LIN {X 0,Y 599.988,Z 849.399,A -85,B 0,C 180,E1 26596.435,E2 26596.435} C_VEL
LIN {X 0,Y 597.537,Z 878.172,A -85,B 0,C 180,E1 26595.722,E2 26595.722} C_VEL
LIN {X 0,Y 595.265,Z 899.969,A -85,B 0,C 180,E1 26595.037,E2 26595.037} C_VEL
LIN {X 0,Y 592.79,Z 920.942,A -85,B 0,C 180,E1 26594.253,E2 26594.253} C_VEL
LIN {X 0,Y 590.222,Z 940.863,A -85,B 0,C 180,E1 26593.384,E2 26593.384} C_VEL
LIN {X 0,Y 587.234,Z 961.854,A -85,B 0,C 180,E1 26592.336,E2 26592.336} C_VEL
LIN {X 0,Y 583.301,Z 987.615,A -85,B 0,C 180,E1 26590.839,E2 26590.839} C_VEL
LIN {X 0,Y 579.885,Z 1008.289,A -85,B 0,C 180,E1 26589.448,E2 26589.448} C_VEL
LIN {X 0,Y 576.852,Z 1026.156,A -85,B 0,C 180,E1 26588.099,E2 26588.099} C_VEL
LIN {X 0,Y 574.033,Z 1042.219,A -85,B 0,C 180,E1 26586.749,E2 26586.749} C_VEL
LIN {X 0,Y 571.11,Z 1058.494,A -85,B 0,C 180,E1 26585.23,E2 26585.23} C_VEL
LIN {X 0,Y 568.193,Z 1074.819,A -85,B 0,C 180,E1 26583.542,E2 26583.542} C_VEL
LIN {X 0,Y 564.878,Z 1093.745,A -85,B 0,C 180,E1 26581.358,E2 26581.358} C_VEL
LIN {X 0,Y 561.877,Z 1111.065,A -85,B 0,C 180,E1 26579.065,E2 26579.065} C_VEL
LIN {X 0,Y 559.756,Z 1124.375,A -85,B 0,C 180,E1 26577.096,E2 26577.096} C_VEL
LIN {X 0,Y 557.748,Z 1137.63,A -85,B 0,C 180,E1 26574.915,E2 26574.915} C_VEL
LIN {X 0,Y 555.8,Z 1152.163,A -85,B 0,C 180,E1 26572.196,E2 26572.196} C_VEL
LIN {X 0,Y 554.441,Z 1163.606,A -85,B 0,C 180,E1 26569.708,E2 26569.708} C_VEL
LIN {X 0,Y 553.521,Z 1172.704,A -85,B 0,C 180,E1 26567.449,E2 26567.449} C_VEL
LIN {X 0,Y 552.864,Z 1180.922,A -85,B 0,C 180,E1 26565.095,E2 26565.095} C_VEL
LIN {X 0,Y 552.339,Z 1189.025,A -85,B 0,C 180,E1 26562.334,E2 26562.334} C_VEL
LIN {X 0,Y 552.078,Z 1195.294,A -85,B 0,C 180,E1 26559.591,E2 26559.591} C_VEL
LIN {X 0,Y 551.97,Z 1199.532,A -85,B 0,C 180,E1 26557.18,E2 26557.18} C_VEL
LIN {X 0,Y 551.918,Z 1202.669,A -85,B 0,C 180,E1 26554.676,E2 26554.676} C_VEL
LIN {X 0,Y 551.91,Z 1204.6,A -85,B 0,C 180,E1 26551.869,E2 26551.869} C_VEL
LIN {X 0,Y 551.895,Z 1204.872,A -85,B 0,C 180,E1 26549.377,E2 26549.377} C_VEL
LIN {X 0,Y 551.916,Z 1203.978,A -85,B 0,C 180,E1 26546.988,E2 26546.988} C_VEL
LIN {X 0,Y 551.93,Z 1201.872,A -85,B 0,C 180,E1 26544.595,E2 26544.595} C_VEL
LIN {X 0,Y 552,Z 1198.251,A -85,B 0,C 180,E1 26541.983,E2 26541.983} C_VEL
LIN {X 0,Y 552.17,Z 1192.609,A -85,B 0,C 180,E1 26539.145,E2 26539.145} C_VEL
LIN {X 0,Y 552.519,Z 1186.072,A -85,B 0,C 180,E1 26536.607,E2 26536.607} C_VEL
LIN {X 0,Y 552.999,Z 1178.8,A -85,B 0,C 180,E1 26534.264,E2 26534.264} C_VEL
LIN {X 0,Y 553.836,Z 1169.631,A -85,B 0,C 180,E1 26531.739,E2 26531.739} C_VEL
LIN {X 0,Y 555.152,Z 1157.326,A -85,B 0,C 180,E1 26528.887,E2 26528.887} C_VEL
LIN {X 0,Y 556.58,Z 1145.997,A -85,B 0,C 180,E1 26526.609,E2 26526.609} C_VEL
LIN {X 0,Y 558.321,Z 1133.823,A -85,B 0,C 180,E1 26524.432,E2 26524.432} C_VEL
LIN {X 0,Y 560.9,Z 1117.228,A -85,B 0,C 180,E1 26521.811,E2 26521.811} C_VEL
LIN {X 0,Y 563.604,Z 1100.917,A -85,B 0,C 180,E1 26519.567,E2 26519.567} C_VEL
LIN {X 0,Y 566.273,Z 1085.443,A -85,B 0,C 180,E1 26517.656,E2 26517.656} C_VEL
LIN {X 0,Y 569.654,Z 1066.711,A -85,B 0,C 180,E1 26515.586,E2 26515.586} C_VEL
LIN {X 0,Y 573.385,Z 1045.863,A -85,B 0,C 180,E1 26513.576,E2 26513.576} C_VEL
LIN {X 0,Y 576.391,Z 1028.822,A -85,B 0,C 180,E1 26512.115,E2 26512.115} C_VEL
LIN {X 0,Y 579.366,Z 1011.299,A -85,B 0,C 180,E1 26510.77,E2 26510.77} C_VEL
LIN {X 0,Y 582.452,Z 992.608,A -85,B 0,C 180,E1 26509.484,E2 26509.484} C_VEL
LIN {X 0,Y 585.633,Z 972.478,A -85,B 0,C 180,E1 26508.253,E2 26508.253} C_VEL
LIN {X 0,Y 589.484,Z 946.5,A -85,B 0,C 180,E1 26506.878,E2 26506.878} C_VEL
LIN {X 0,Y 592.403,Z 924.112,A -85,B 0,C 180,E1 26505.876,E2 26505.876} C_VEL
LIN {X 0,Y 594.962,Z 902.704,A -85,B 0,C 180,E1 26505.059,E2 26505.059} C_VEL
LIN {X 0,Y 597.166,Z 881.774,A -85,B 0,C 180,E1 26504.383,E2 26504.383} C_VEL
LIN {X 0,Y 599.156,Z 859.782,A -85,B 0,C 180,E1 26503.799,E2 26503.799} C_VEL
LIN {X 0,Y 601.177,Z 832.126,A -85,B 0,C 180,E1 26503.233,E2 26503.233} C_VEL
LIN {X 0,Y 602.837,Z 786.304,A -85,B 0,C 180,E1 26502.56,E2 26502.56} C_VEL
LIN {X 0,Y 609.733,Z 564.773,A -85,B 0,C 180,E1 26499.403,E2 26499.403} C_VEL
LIN {X 0,Y 614.382,Z 422.014,A -85,B 0,C 180,E1 26497.318,E2 26497.318} C_VEL
LIN {X 0,Y 602.713,Z 404.172,A -85,B 0,C 180,E1 26495.496,E2 26495.496} C_VEL
LIN {X 0,Y 590.418,Z 386.403,A -85,B 0,C 180,E1 26493.424,E2 26493.424} C_VEL
LIN {X 0,Y 579.878,Z 372.071,A -85,B 0,C 180,E1 26491.498,E2 26491.498} C_VEL
LIN {X 0,Y 572.08,Z 361.83,A -85,B 0,C 180,E1 26489.963,E2 26489.963} C_VEL
LIN {X 0,Y 567.6,Z 356.163,A -85,B 0,C 180,E1 26489.034,E2 26489.034} C_VEL
LIN {X 0,Y 563.365,Z 350.725,A -85,B 0,C 180,E1 26488.114,E2 26488.114} C_VEL
LIN {X 0,Y 559.96,Z 346.445,A -85,B 0,C 180,E1 26487.346,E2 26487.346} C_VEL
LIN {X 0,Y 557.435,Z 343.483,A -85,B 0,C 180,E1 26486.716,E2 26486.716} C_VEL
LIN {X 0,Y 555.888,Z 340.01,A -85,B 0,C 180,E1 26485.919,E2 26485.919} C_VEL
LIN {X 0,Y 553.761,Z 336.637,A -85,B 0,C 180,E1 26484.988,E2 26484.988} C_VEL
LIN {X 0,Y 553.461,Z 335.24,A -85,B 0,C 180,E1 26484.666,E2 26484.666} C_VEL
LIN {X 0,Y 553.477,Z 335.245,A -85,B 0,C 180,E1 26481.292,E2 26481.292} C_VEL
LIN {X 0,Y 553.497,Z 335.282,A -85,B 0,C 180,E1 26477.994,E2 26477.994} C_VEL
LIN {X 0,Y 553.448,Z 335.235,A -85,B 0,C 180,E1 26474.758,E2 26474.758} C_VEL
LIN {X 0,Y 553.503,Z 335.278,A -85,B 0,C 180,E1 26471.462,E2 26471.462} C_VEL
LIN {X 0,Y 553.449,Z 335.241,A -85,B 0,C 180,E1 26468.206,E2 26468.206} C_VEL
LIN {X 0,Y 553.46,Z 335.263,A -85,B 0,C 180,E1 26464.871,E2 26464.871} C_VEL
LIN {X 0,Y 553.478,Z 335.25,A -85,B 0,C 180,E1 26461.656,E2 26461.656} C_VEL
LIN {X 0,Y 553.437,Z 335.255,A -85,B 0,C 180,E1 26458.447,E2 26458.447} C_VEL
LIN {X 0,Y 553.498,Z 335.258,A -85,B 0,C 180,E1 26455.233,E2 26455.233} C_VEL
LIN {X 0,Y 553.429,Z 335.249,A -85,B 0,C 180,E1 26452.108,E2 26452.108} C_VEL
LIN {X 0,Y 553.481,Z 335.272,A -85,B 0,C 180,E1 26448.854,E2 26448.854} C_VEL
LIN {X 0,Y 553.424,Z 335.242,A -85,B 0,C 180,E1 26445.776,E2 26445.776} C_VEL
LIN {X 0,Y 553.45,Z 335.293,A -85,B 0,C 180,E1 26442.44,E2 26442.44} C_VEL
LIN {X 0,Y 553.434,Z 335.237,A -85,B 0,C 180,E1 26439.364,E2 26439.364} C_VEL
LIN {X 0,Y 553.421,Z 335.272,A -85,B 0,C 180,E1 26436.014,E2 26436.014} C_VEL
LIN {X 0,Y 553.44,Z 335.455,A -85,B 0,C 180,E1 26433.785,E2 26433.785} C_VEL
LIN {X 0,Y 554.447,Z 338.299,A -85,B 0,C 180,E1 26433.491,E2 26433.491} C_VEL
LIN {X 0,Y 556.848,Z 340.849,A -85,B 0,C 180,E1 26432.923,E2 26432.923} C_VEL
LIN {X 0,Y 558.75,Z 342.157,A -85,B 0,C 180,E1 26432.503,E2 26432.503} C_VEL
LIN {X 0,Y 560.898,Z 345.768,A -85,B 0,C 180,E1 26431.983,E2 26431.983} C_VEL
LIN {X 0,Y 564.13,Z 348.556,A -85,B 0,C 180,E1 26431.293,E2 26431.293} C_VEL
LIN {X 0,Y 566.949,Z 352.543,A -85,B 0,C 180,E1 26430.669,E2 26430.669} C_VEL
LIN {X 0,Y 569.277,Z 354.812,A -85,B 0,C 180,E1 26430.194,E2 26430.194} C_VEL
LIN {X 0,Y 572.686,Z 359.091,A -85,B 0,C 180,E1 26429.493,E2 26429.493} C_VEL
LIN {X 0,Y 574.265,Z 360.906,A -85,B 0,C 180,E1 26429.18,E2 26429.18} C_VEL
LIN {X 0,Y 578.146,Z 365.563,A -85,B 0,C 180,E1 26428.426,E2 26428.426} C_VEL
LIN {X 0,Y 584.331,Z 373.412,A -85,B 0,C 180,E1 26427.266,E2 26427.266} C_VEL
LIN {X 0,Y 591.597,Z 382.48,A -85,B 0,C 180,E1 26425.983,E2 26425.983} C_VEL
LIN {X 0,Y 603.802,Z 398.638,A -85,B 0,C 180,E1 26423.964,E2 26423.964} C_VEL
LIN {X 0,Y 614.272,Z 413.349,A -85,B 0,C 180,E1 26422.352,E2 26422.352} C_VEL
LIN {X 0,Y 607.005,Z 631.906,A -85,B 0,C 180,E1 26419.19,E2 26419.19} C_VEL
LIN {X 0,Y 603.673,Z 738.694,A -85,B 0,C 180,E1 26417.669,E2 26417.669} C_VEL
LIN {X 0,Y 602.74,Z 746.4,A -85,B 0,C 180,E1 26417.633,E2 26417.633} C_VEL
LIN {X 0,Y 597.897,Z 767.028,A -85,B 0,C 180,E1 26417.785,E2 26417.785} C_VEL
LIN {X 0,Y 597.208,Z 773.633,A -85,B 0,C 180,E1 26417.742,E2 26417.742} C_VEL
LIN {X 0,Y 595.598,Z 809.869,A -85,B 0,C 180,E1 26417.181,E2 26417.181} C_VEL
LIN {X 0,Y 593.757,Z 833.921,A -85,B 0,C 180,E1 26416.665,E2 26416.665} C_VEL
LIN {X 0,Y 591.733,Z 855.327,A -85,B 0,C 180,E1 26416.083,E2 26416.083} C_VEL
LIN {X 0,Y 589.538,Z 875.33,A -85,B 0,C 180,E1 26415.424,E2 26415.424} C_VEL
LIN {X 0,Y 586.99,Z 895.612,A -85,B 0,C 180,E1 26414.639,E2 26414.639} C_VEL
LIN {X 0,Y 583.725,Z 919.209,A -85,B 0,C 180,E1 26413.566,E2 26413.566} C_VEL
LIN {X 0,Y 579.717,Z 944.344,A -85,B 0,C 180,E1 26412.205,E2 26412.205} C_VEL
LIN {X 0,Y 576.363,Z 963.977,A -85,B 0,C 180,E1 26410.976,E2 26410.976} C_VEL
LIN {X 0,Y 573.108,Z 982.083,A -85,B 0,C 180,E1 26409.699,E2 26409.699} C_VEL
LIN {X 0,Y 569.76,Z 1000.085,A -85,B 0,C 180,E1 26408.277,E2 26408.277} C_VEL
LIN {X 0,Y 565.664,Z 1021.503,A -85,B 0,C 180,E1 26406.372,E2 26406.372} C_VEL
LIN {X 0,Y 561.8,Z 1041.554,A -85,B 0,C 180,E1 26404.327,E2 26404.327} C_VEL
LIN {X 0,Y 558.837,Z 1057.414,A -85,B 0,C 180,E1 26402.523,E2 26402.523} C_VEL
LIN {X 0,Y 555.913,Z 1073.578,A -85,B 0,C 180,E1 26400.478,E2 26400.478} C_VEL
LIN {X 0,Y 552.664,Z 1092.003,A -85,B 0,C 180,E1 26397.824,E2 26397.824} C_VEL
LIN {X 0,Y 550.501,Z 1105.479,A -85,B 0,C 180,E1 26395.612,E2 26395.612} C_VEL
LIN {X 0,Y 548.641,Z 1118.062,A -85,B 0,C 180,E1 26393.295,E2 26393.295} C_VEL
LIN {X 0,Y 546.895,Z 1131.586,A -85,B 0,C 180,E1 26390.438,E2 26390.438} C_VEL
LIN {X 0,Y 545.756,Z 1141.728,A -85,B 0,C 180,E1 26387.926,E2 26387.926} C_VEL
LIN {X 0,Y 545.016,Z 1149.714,A -85,B 0,C 180,E1 26385.645,E2 26385.645} C_VEL
LIN {X 0,Y 544.517,Z 1156.853,A -85,B 0,C 180,E1 26383.269,E2 26383.269} C_VEL
LIN {X 0,Y 544.153,Z 1163.946,A -85,B 0,C 180,E1 26380.374,E2 26380.374} C_VEL
LIN {X 0,Y 543.987,Z 1168.822,A -85,B 0,C 180,E1 26377.711,E2 26377.711} C_VEL
LIN {X 0,Y 543.928,Z 1172.048,A -85,B 0,C 180,E1 26375.274,E2 26375.274} C_VEL
LIN {X 0,Y 543.911,Z 1174.082,A -85,B 0,C 180,E1 26372.845,E2 26372.845} C_VEL
LIN {X 0,Y 543.907,Z 1174.974,A -85,B 0,C 180,E1 26370.105,E2 26370.105} C_VEL
LIN {X 0,Y 543.908,Z 1174.209,A -85,B 0,C 180,E1 26367.26,E2 26367.26} C_VEL
LIN {X 0,Y 543.924,Z 1172.26,A -85,B 0,C 180,E1 26364.832,E2 26364.832} C_VEL
LIN {X 0,Y 543.974,Z 1169.277,A -85,B 0,C 180,E1 26362.501,E2 26362.501} C_VEL
LIN {X 0,Y 544.103,Z 1164.965,A -85,B 0,C 180,E1 26360.053,E2 26360.053} C_VEL
LIN {X 0,Y 544.431,Z 1158.303,A -85,B 0,C 180,E1 26357.161,E2 26357.161} C_VEL
LIN {X 0,Y 544.968,Z 1150.36,A -85,B 0,C 180,E1 26354.463,E2 26354.463} C_VEL
LIN {X 0,Y 545.681,Z 1142.463,A -85,B 0,C 180,E1 26352.182,E2 26352.182} C_VEL
LIN {X 0,Y 546.677,Z 1133.331,A -85,B 0,C 180,E1 26349.889,E2 26349.889} C_VEL
LIN {X 0,Y 548.28,Z 1120.798,A -85,B 0,C 180,E1 26347.143,E2 26347.143} C_VEL
LIN {X 0,Y 550.321,Z 1106.606,A -85,B 0,C 180,E1 26344.495,E2 26344.495} C_VEL
LIN {X 0,Y 552.349,Z 1093.942,A -85,B 0,C 180,E1 26342.393,E2 26342.393} C_VEL
LIN {X 0,Y 554.911,Z 1079.043,A -85,B 0,C 180,E1 26340.178,E2 26340.178} C_VEL
LIN {X 0,Y 558.47,Z 1059.488,A -85,B 0,C 180,E1 26337.635,E2 26337.635} C_VEL
LIN {X 0,Y 561.504,Z 1043.16,A -85,B 0,C 180,E1 26335.758,E2 26335.758} C_VEL
LIN {X 0,Y 564.674,Z 1026.355,A -85,B 0,C 180,E1 26334.021,E2 26334.021} C_VEL
LIN {X 0,Y 568.677,Z 1005.892,A -85,B 0,C 180,E1 26332.114,E2 26332.114} C_VEL
LIN {X 0,Y 572.798,Z 983.808,A -85,B 0,C 180,E1 26330.338,E2 26330.338} C_VEL
LIN {X 0,Y 576.126,Z 965.309,A -85,B 0,C 180,E1 26329.022,E2 26329.022} C_VEL
LIN {X 0,Y 579.352,Z 946.439,A -85,B 0,C 180,E1 26327.829,E2 26327.829} C_VEL
LIN {X 0,Y 582.723,Z 925.413,A -85,B 0,C 180,E1 26326.66,E2 26326.66} C_VEL
LIN {X 0,Y 586.616,Z 898.562,A -85,B 0,C 180,E1 26325.394,E2 26325.394} C_VEL
LIN {X 0,Y 589.41,Z 876.434,A -85,B 0,C 180,E1 26324.525,E2 26324.525} C_VEL
LIN {X 0,Y 591.727,Z 855.412,A -85,B 0,C 180,E1 26323.83,E2 26323.83} C_VEL
LIN {X 0,Y 593.743,Z 834.118,A -85,B 0,C 180,E1 26323.251,E2 26323.251} C_VEL
LIN {X 0,Y 595.557,Z 810.404,A -85,B 0,C 180,E1 26322.74,E2 26322.74} C_VEL
LIN {X 0,Y 597.184,Z 774.353,A -85,B 0,C 180,E1 26322.178,E2 26322.178} C_VEL
LIN {X 0,Y 604.577,Z 550.918,A -85,B 0,C 180,E1 26318.968,E2 26318.968} C_VEL
LIN {X 0,Y 609.231,Z 417.375,A -85,B 0,C 180,E1 26317.008,E2 26317.008} C_VEL
LIN {X 0,Y 597.885,Z 401.698,A -85,B 0,C 180,E1 26315.209,E2 26315.209} C_VEL
LIN {X 0,Y 587.512,Z 387.83,A -85,B 0,C 180,E1 26313.435,E2 26313.435} C_VEL
LIN {X 0,Y 578.153,Z 376.088,A -85,B 0,C 180,E1 26311.719,E2 26311.719} C_VEL
LIN {X 0,Y 574.829,Z 371.978,A -85,B 0,C 180,E1 26311.077,E2 26311.077} C_VEL
LIN {X 0,Y 570.013,Z 366.1,A -85,B 0,C 180,E1 26310.112,E2 26310.112} C_VEL
LIN {X 0,Y 565.664,Z 360.778,A -85,B 0,C 180,E1 26309.201,E2 26309.201} C_VEL
LIN {X 0,Y 562.258,Z 356.818,A -85,B 0,C 180,E1 26308.464,E2 26308.464} C_VEL
LIN {X 0,Y 561.023,Z 355.163,A -85,B 0,C 180,E1 26308.184,E2 26308.184} C_VEL
LIN {X 0,Y 557.676,Z 351.854,A -85,B 0,C 180,E1 26307.438,E2 26307.438} C_VEL
LIN {X 0,Y 555.938,Z 349.05,A -85,B 0,C 180,E1 26307.01,E2 26307.01} C_VEL
LIN {X 0,Y 552.681,Z 346.292,A -85,B 0,C 180,E1 26306.253,E2 26306.253} C_VEL
LIN {X 0,Y 550.679,Z 342.754,A -85,B 0,C 180,E1 26305.719,E2 26305.719} C_VEL
LIN {X 0,Y 547.427,Z 340.512,A -85,B 0,C 180,E1 26304.928,E2 26304.928} C_VEL
LIN {X 0,Y 545.843,Z 337.847,A -85,B 0,C 180,E1 26304.481,E2 26304.481} C_VEL
LIN {X 0,Y 545.469,Z 336.245,A -85,B 0,C 180,E1 26304.33,E2 26304.33} C_VEL
LIN {X 0,Y 545.544,Z 336.224,A -85,B 0,C 180,E1 26301.166,E2 26301.166} C_VEL
LIN {X 0,Y 545.481,Z 336.282,A -85,B 0,C 180,E1 26297.936,E2 26297.936} C_VEL
LIN {X 0,Y 545.505,Z 336.221,A -85,B 0,C 180,E1 26294.586,E2 26294.586} C_VEL
LIN {X 0,Y 545.5,Z 336.281,A -85,B 0,C 180,E1 26291.525,E2 26291.525} C_VEL
LIN {X 0,Y 545.489,Z 336.226,A -85,B 0,C 180,E1 26288.114,E2 26288.114} C_VEL
LIN {X 0,Y 545.536,Z 336.265,A -85,B 0,C 180,E1 26285.047,E2 26285.047} C_VEL
LIN {X 0,Y 545.491,Z 336.229,A -85,B 0,C 180,E1 26281.786,E2 26281.786} C_VEL
LIN {X 0,Y 545.563,Z 336.252,A -85,B 0,C 180,E1 26278.635,E2 26278.635} C_VEL
LIN {X 0,Y 545.5,Z 336.235,A -85,B 0,C 180,E1 26275.374,E2 26275.374} C_VEL
LIN {X 0,Y 545.534,Z 336.236,A -85,B 0,C 180,E1 26272.099,E2 26272.099} C_VEL
LIN {X 0,Y 545.528,Z 336.251,A -85,B 0,C 180,E1 26268.904,E2 26268.904} C_VEL
LIN {X 0,Y 545.511,Z 336.224,A -85,B 0,C 180,E1 26265.565,E2 26265.565} C_VEL
LIN {X 0,Y 545.568,Z 336.274,A -85,B 0,C 180,E1 26262.288,E2 26262.288} C_VEL
LIN {X 0,Y 545.519,Z 336.229,A -85,B 0,C 180,E1 26258.946,E2 26258.946} C_VEL
LIN {X 0,Y 545.535,Z 336.344,A -85,B 0,C 180,E1 26256.906,E2 26256.906} C_VEL
LIN {X 0,Y 546.888,Z 339.751,A -85,B 0,C 180,E1 26256.053,E2 26256.053} C_VEL
LIN {X 0,Y 548.427,Z 341.539,A -85,B 0,C 180,E1 26255.437,E2 26255.437} C_VEL
LIN {X 0,Y 549.416,Z 343.962,A -85,B 0,C 180,E1 26254.939,E2 26254.939} C_VEL
LIN {X 0,Y 553.071,Z 348.19,A -85,B 0,C 180,E1 26254.026,E2 26254.026} C_VEL
LIN {X 0,Y 557.925,Z 354.223,A -85,B 0,C 180,E1 26252.864,E2 26252.864} C_VEL
LIN {X 0,Y 562.346,Z 359.743,A -85,B 0,C 180,E1 26251.859,E2 26251.859} C_VEL
LIN {X 0,Y 567.765,Z 366.71,A -85,B 0,C 180,E1 26250.686,E2 26250.686} C_VEL
LIN {X 0,Y 574.835,Z 376.016,A -85,B 0,C 180,E1 26249.243,E2 26249.243} C_VEL
LIN {X 0,Y 584.56,Z 389.121,A -85,B 0,C 180,E1 26247.397,E2 26247.397} C_VEL
LIN {X 0,Y 597.209,Z 407.344,A -85,B 0,C 180,E1 26245.185,E2 26245.185} C_VEL
LIN {X 0,Y 608.535,Z 424.744,A -85,B 0,C 180,E1 26243.354,E2 26243.354} C_VEL
LIN {X 0,Y 609.46,Z 426.604,A -85,B 0,C 180,E1 26243.203,E2 26243.203} C_VEL
LIN {X 0,Y 602.086,Z 641.22,A -85,B 0,C 180,E1 26240.079,E2 26240.079} C_VEL
LIN {X 0,Y 596.02,Z 824.957,A -85,B 0,C 180,E1 26237.439,E2 26237.439} C_VEL
LIN {X 0,Y 594.452,Z 849.135,A -85,B 0,C 180,E1 26236.999,E2 26236.999} C_VEL
LIN {X 0,Y 591.903,Z 877.906,A -85,B 0,C 180,E1 26236.284,E2 26236.284} C_VEL
LIN {X 0,Y 589.532,Z 899.701,A -85,B 0,C 180,E1 26235.598,E2 26235.598} C_VEL
LIN {X 0,Y 587.049,Z 919.963,A -85,B 0,C 180,E1 26234.839,E2 26234.839} C_VEL
LIN {X 0,Y 584.431,Z 939.39,A -85,B 0,C 180,E1 26233.995,E2 26233.995} C_VEL
LIN {X 0,Y 581.418,Z 959.656,A -85,B 0,C 180,E1 26232.989,E2 26232.989} C_VEL
LIN {X 0,Y 577.606,Z 983.983,A -85,B 0,C 180,E1 26231.597,E2 26231.597} C_VEL
LIN {X 0,Y 573.59,Z 1007.265,A -85,B 0,C 180,E1 26230.033,E2 26230.033} C_VEL
LIN {X 0,Y 570.275,Z 1025.853,A -85,B 0,C 180,E1 26228.621,E2 26228.621} C_VEL
LIN {X 0,Y 567.138,Z 1043.078,A -85,B 0,C 180,E1 26227.165,E2 26227.165} C_VEL
LIN {X 0,Y 564.18,Z 1059.048,A -85,B 0,C 180,E1 26225.666,E2 26225.666} C_VEL
LIN {X 0,Y 560.905,Z 1076.539,A -85,B 0,C 180,E1 26223.828,E2 26223.828} C_VEL
LIN {X 0,Y 557.046,Z 1097.135,A -85,B 0,C 180,E1 26221.368,E2 26221.368} C_VEL
LIN {X 0,Y 554.404,Z 1111.834,A -85,B 0,C 180,E1 26219.376,E2 26219.376} C_VEL
LIN {X 0,Y 552.177,Z 1125.074,A -85,B 0,C 180,E1 26217.383,E2 26217.383} C_VEL
LIN {X 0,Y 549.977,Z 1138.898,A -85,B 0,C 180,E1 26215.062,E2 26215.062} C_VEL
LIN {X 0,Y 547.867,Z 1153.716,A -85,B 0,C 180,E1 26212.196,E2 26212.196} C_VEL
LIN {X 0,Y 546.577,Z 1164.063,A -85,B 0,C 180,E1 26209.892,E2 26209.892} C_VEL
LIN {X 0,Y 545.609,Z 1173.108,A -85,B 0,C 180,E1 26207.6,E2 26207.6} C_VEL
LIN {X 0,Y 544.864,Z 1181.98,A -85,B 0,C 180,E1 26204.995,E2 26204.995} C_VEL
LIN {X 0,Y 544.319,Z 1190.062,A -85,B 0,C 180,E1 26202.088,E2 26202.088} C_VEL
LIN {X 0,Y 544.084,Z 1195.498,A -85,B 0,C 180,E1 26199.627,E2 26199.627} C_VEL
LIN {X 0,Y 543.976,Z 1199.529,A -85,B 0,C 180,E1 26197.286,E2 26197.286} C_VEL
LIN {X 0,Y 543.919,Z 1202.666,A -85,B 0,C 180,E1 26194.745,E2 26194.745} C_VEL
LIN {X 0,Y 543.91,Z 1204.6,A -85,B 0,C 180,E1 26191.896,E2 26191.896} C_VEL
LIN {X 0,Y 543.895,Z 1204.872,A -85,B 0,C 180,E1 26189.368,E2 26189.368} C_VEL
LIN {X 0,Y 543.915,Z 1204.043,A -85,B 0,C 180,E1 26187.05,E2 26187.05} C_VEL
LIN {X 0,Y 543.93,Z 1202.097,A -85,B 0,C 180,E1 26184.726,E2 26184.726} C_VEL
LIN {X 0,Y 543.982,Z 1198.889,A -85,B 0,C 180,E1 26182.289,E2 26182.289} C_VEL
LIN {X 0,Y 544.153,Z 1193.818,A -85,B 0,C 180,E1 26179.519,E2 26179.519} C_VEL
LIN {X 0,Y 544.513,Z 1186.94,A -85,B 0,C 180,E1 26176.717,E2 26176.717} C_VEL
LIN {X 0,Y 545.002,Z 1179.859,A -85,B 0,C 180,E1 26174.355,E2 26174.355} C_VEL
LIN {X 0,Y 545.737,Z 1171.893,A -85,B 0,C 180,E1 26172.074,E2 26172.074} C_VEL
LIN {X 0,Y 546.863,Z 1161.773,A -85,B 0,C 180,E1 26169.561,E2 26169.561} C_VEL
LIN {X 0,Y 548.605,Z 1148.289,A -85,B 0,C 180,E1 26166.703,E2 26166.703} C_VEL
LIN {X 0,Y 550.465,Z 1135.727,A -85,B 0,C 180,E1 26164.386,E2 26164.386} C_VEL
LIN {X 0,Y 552.556,Z 1122.677,A -85,B 0,C 180,E1 26162.237,E2 26162.237} C_VEL
LIN {X 0,Y 555.576,Z 1105.587,A -85,B 0,C 180,E1 26159.741,E2 26159.741} C_VEL
LIN {X 0,Y 558.686,Z 1088.219,A -85,B 0,C 180,E1 26157.527,E2 26157.527} C_VEL
LIN {X 0,Y 561.576,Z 1072.791,A -85,B 0,C 180,E1 26155.763,E2 26155.763} C_VEL
LIN {X 0,Y 564.688,Z 1056.271,A -85,B 0,C 180,E1 26154.058,E2 26154.058} C_VEL
LIN {X 0,Y 568.601,Z 1035.264,A -85,B 0,C 180,E1 26152.143,E2 26152.143} C_VEL
LIN {X 0,Y 572.64,Z 1012.608,A -85,B 0,C 180,E1 26150.357,E2 26150.357} C_VEL
LIN {X 0,Y 575.879,Z 993.922,A -85,B 0,C 180,E1 26149.051,E2 26149.051} C_VEL
LIN {X 0,Y 579.022,Z 974.931,A -85,B 0,C 180,E1 26147.866,E2 26147.866} C_VEL
LIN {X 0,Y 582.24,Z 954.318,A -85,B 0,C 180,E1 26146.731,E2 26146.731} C_VEL
LIN {X 0,Y 586.071,Z 927.723,A -85,B 0,C 180,E1 26145.478,E2 26145.478} C_VEL
LIN {X 0,Y 589.019,Z 904.168,A -85,B 0,C 180,E1 26144.56,E2 26144.56} C_VEL
LIN {X 0,Y 591.374,Z 882.88,A -85,B 0,C 180,E1 26143.862,E2 26143.862} C_VEL
LIN {X 0,Y 593.406,Z 861.558,A -85,B 0,C 180,E1 26143.285,E2 26143.285} C_VEL
LIN {X 0,Y 595.218,Z 838.552,A -85,B 0,C 180,E1 26142.793,E2 26142.793} C_VEL
LIN {X 0,Y 596.91,Z 802.56,A -85,B 0,C 180,E1 26142.227,E2 26142.227} C_VEL
LIN {X 0,Y 604.236,Z 576.787,A -85,B 0,C 180,E1 26138.991,E2 26138.991} C_VEL
LIN {X 0,Y 609.363,Z 426.095,A -85,B 0,C 180,E1 26136.778,E2 26136.778} C_VEL
LIN {X 0,Y 598.955,Z 410.049,A -85,B 0,C 180,E1 26135.113,E2 26135.113} C_VEL
LIN {X 0,Y 587.138,Z 392.817,A -85,B 0,C 180,E1 26133.08,E2 26133.08} C_VEL
LIN {X 0,Y 576.945,Z 378.813,A -85,B 0,C 180,E1 26131.182,E2 26131.182} C_VEL
LIN {X 0,Y 569.231,Z 368.59,A -85,B 0,C 180,E1 26129.635,E2 26129.635} C_VEL
LIN {X 0,Y 564.802,Z 362.949,A -85,B 0,C 180,E1 26128.699,E2 26128.699} C_VEL
LIN {X 0,Y 560.615,Z 357.563,A -85,B 0,C 180,E1 26127.772,E2 26127.772} C_VEL
LIN {X 0,Y 555.841,Z 351.649,A -85,B 0,C 180,E1 26126.668,E2 26126.668} C_VEL
LIN {X 0,Y 551.729,Z 346.574,A -85,B 0,C 180,E1 26125.667,E2 26125.667} C_VEL
LIN {X 0,Y 548.782,Z 342.824,A -85,B 0,C 180,E1 26124.861,E2 26124.861} C_VEL
LIN {X 0,Y 548.051,Z 341.123,A -85,B 0,C 180,E1 26124.444,E2 26124.444} C_VEL
LIN {X 0,Y 545.848,Z 337.649,A -85,B 0,C 180,E1 26123.407,E2 26123.407} C_VEL
LIN {X 0,Y 545.527,Z 336.271,A -85,B 0,C 180,E1 26123.063,E2 26123.063} C_VEL
LIN {X 0,Y 545.562,Z 336.219,A -85,B 0,C 180,E1 26119.82,E2 26119.82} C_VEL
LIN {X 0,Y 545.518,Z 336.251,A -85,B 0,C 180,E1 26116.548,E2 26116.548} C_VEL
LIN {X 0,Y 545.543,Z 336.243,A -85,B 0,C 180,E1 26113.244,E2 26113.244} C_VEL
LIN {X 0,Y 545.528,Z 336.226,A -85,B 0,C 180,E1 26110.028,E2 26110.028} C_VEL
LIN {X 0,Y 545.512,Z 336.274,A -85,B 0,C 180,E1 26106.631,E2 26106.631} C_VEL
LIN {X 0,Y 545.555,Z 336.213,A -85,B 0,C 180,E1 26103.362,E2 26103.362} C_VEL
LIN {X 0,Y 545.507,Z 336.28,A -85,B 0,C 180,E1 26100.105,E2 26100.105} C_VEL
LIN {X 0,Y 545.514,Z 336.218,A -85,B 0,C 180,E1 26096.743,E2 26096.743} C_VEL
LIN {X 0,Y 545.525,Z 336.277,A -85,B 0,C 180,E1 26093.58,E2 26093.58} C_VEL
LIN {X 0,Y 545.49,Z 336.226,A -85,B 0,C 180,E1 26090.291,E2 26090.291} C_VEL
LIN {X 0,Y 545.554,Z 336.257,A -85,B 0,C 180,E1 26087.079,E2 26087.079} C_VEL
LIN {X 0,Y 545.481,Z 336.237,A -85,B 0,C 180,E1 26083.931,E2 26083.931} C_VEL
LIN {X 0,Y 545.538,Z 336.234,A -85,B 0,C 180,E1 26080.715,E2 26080.715} C_VEL
LIN {X 0,Y 545.483,Z 336.263,A -85,B 0,C 180,E1 26077.587,E2 26077.587} C_VEL
LIN {X 0,Y 545.494,Z 336.367,A -85,B 0,C 180,E1 26075.527,E2 26075.527} C_VEL
LIN {X 0,Y 546.426,Z 339.109,A -85,B 0,C 180,E1 26075.226,E2 26075.226} C_VEL
LIN {X 0,Y 548.86,Z 341.772,A -85,B 0,C 180,E1 26074.594,E2 26074.594} C_VEL
LIN {X 0,Y 550.913,Z 343.076,A -85,B 0,C 180,E1 26074.105,E2 26074.105} C_VEL
LIN {X 0,Y 552.978,Z 346.642,A -85,B 0,C 180,E1 26073.559,E2 26073.559} C_VEL
LIN {X 0,Y 556.345,Z 349.597,A -85,B 0,C 180,E1 26072.78,E2 26072.78} C_VEL
LIN {X 0,Y 559.016,Z 353.477,A -85,B 0,C 180,E1 26072.141,E2 26072.141} C_VEL
LIN {X 0,Y 561.68,Z 355.87,A -85,B 0,C 180,E1 26071.563,E2 26071.563} C_VEL
LIN {X 0,Y 564.926,Z 360.122,A -85,B 0,C 180,E1 26070.845,E2 26070.845} C_VEL
LIN {X 0,Y 566.889,Z 362.229,A -85,B 0,C 180,E1 26070.434,E2 26070.434} C_VEL
LIN {X 0,Y 570.743,Z 366.764,A -85,B 0,C 180,E1 26069.64,E2 26069.64} C_VEL
LIN {X 0,Y 575.35,Z 372.494,A -85,B 0,C 180,E1 26068.722,E2 26068.722} C_VEL
LIN {X 0,Y 585.772,Z 385.666,A -85,B 0,C 180,E1 26066.774,E2 26066.774} C_VEL
LIN {X 0,Y 596.595,Z 399.913,A -85,B 0,C 180,E1 26064.91,E2 26064.91} C_VEL
LIN {X 0,Y 608.152,Z 415.934,A -85,B 0,C 180,E1 26063.063,E2 26063.063} C_VEL
LIN {X 0,Y 609.259,Z 417.8,A -85,B 0,C 180,E1 26062.887,E2 26062.887} C_VEL
LIN {X 0,Y 601.72,Z 634.699,A -85,B 0,C 180,E1 26059.731,E2 26059.731} C_VEL
LIN {X 0,Y 597.208,Z 773.633,A -85,B 0,C 180,E1 26057.742,E2 26057.742} C_VEL
LIN {X 0,Y 596.321,Z 781.341,A -85,B 0,C 180,E1 26057.704,E2 26057.704} C_VEL
LIN {X 0,Y 591.261,Z 801.934,A -85,B 0,C 180,E1 26057.849,E2 26057.849} C_VEL
LIN {X 0,Y 590.315,Z 808.486,A -85,B 0,C 180,E1 26057.784,E2 26057.784} C_VEL
LIN {X 0,Y 588.302,Z 833.921,A -85,B 0,C 180,E1 26057.24,E2 26057.24} C_VEL
LIN {X 0,Y 586.207,Z 855.395,A -85,B 0,C 180,E1 26056.655,E2 26056.655} C_VEL
LIN {X 0,Y 583.904,Z 875.613,A -85,B 0,C 180,E1 26055.988,E2 26055.988} C_VEL
LIN {X 0,Y 581.257,Z 895.894,A -85,B 0,C 180,E1 26055.2,E2 26055.2} C_VEL
LIN {X 0,Y 577.896,Z 919.279,A -85,B 0,C 180,E1 26054.131,E2 26054.131} C_VEL
LIN {X 0,Y 573.862,Z 943.732,A -85,B 0,C 180,E1 26052.805,E2 26052.805} C_VEL
LIN {X 0,Y 570.353,Z 963.453,A -85,B 0,C 180,E1 26051.569,E2 26051.569} C_VEL
LIN {X 0,Y 567.044,Z 981.099,A -85,B 0,C 180,E1 26050.325,E2 26050.325} C_VEL
LIN {X 0,Y 563.678,Z 998.386,A -85,B 0,C 180,E1 26048.963,E2 26048.963} C_VEL
LIN {X 0,Y 560.144,Z 1016.079,A -85,B 0,C 180,E1 26047.406,E2 26047.406} C_VEL
LIN {X 0,Y 555.86,Z 1037.235,A -85,B 0,C 180,E1 26045.3,E2 26045.3} C_VEL
LIN {X 0,Y 551.946,Z 1056.492,A -85,B 0,C 180,E1 26043.105,E2 26043.105} C_VEL
LIN {X 0,Y 549.123,Z 1071.047,A -85,B 0,C 180,E1 26041.261,E2 26041.261} C_VEL
LIN {X 0,Y 546.085,Z 1087.705,A -85,B 0,C 180,E1 26038.906,E2 26038.906} C_VEL
LIN {X 0,Y 543.248,Z 1103.662,A -85,B 0,C 180,E1 26036.316,E2 26036.316} C_VEL
LIN {X 0,Y 541.317,Z 1115.771,A -85,B 0,C 180,E1 26034.092,E2 26034.092} C_VEL
LIN {X 0,Y 539.753,Z 1126.611,A -85,B 0,C 180,E1 26031.859,E2 26031.859} C_VEL
LIN {X 0,Y 538.276,Z 1138.464,A -85,B 0,C 180,E1 26029.082,E2 26029.082} C_VEL
LIN {X 0,Y 537.238,Z 1148.302,A -85,B 0,C 180,E1 26026.321,E2 26026.321} C_VEL
LIN {X 0,Y 536.637,Z 1155.687,A -85,B 0,C 180,E1 26023.89,E2 26023.89} C_VEL
LIN {X 0,Y 536.26,Z 1161.734,A -85,B 0,C 180,E1 26021.508,E2 26021.508} C_VEL
LIN {X 0,Y 536.043,Z 1167.264,A -85,B 0,C 180,E1 26018.798,E2 26018.798} C_VEL
LIN {X 0,Y 535.942,Z 1171.478,A -85,B 0,C 180,E1 26015.889,E2 26015.889} C_VEL
LIN {X 0,Y 535.914,Z 1173.807,A -85,B 0,C 180,E1 26013.316,E2 26013.316} C_VEL
LIN {X 0,Y 535.909,Z 1174.771,A -85,B 0,C 180,E1 26011.069,E2 26011.069} C_VEL
LIN {X 0,Y 535.907,Z 1174.791,A -85,B 0,C 180,E1 26008.931,E2 26008.931} C_VEL
LIN {X 0,Y 535.912,Z 1173.865,A -85,B 0,C 180,E1 26006.684,E2 26006.684} C_VEL
LIN {X 0,Y 535.937,Z 1171.688,A -85,B 0,C 180,E1 26004.218,E2 26004.218} C_VEL
LIN {X 0,Y 536.033,Z 1167.706,A -85,B 0,C 180,E1 26001.356,E2 26001.356} C_VEL
LIN {X 0,Y 536.235,Z 1162.199,A -85,B 0,C 180,E1 25998.601,E2 25998.601} C_VEL
LIN {X 0,Y 536.62,Z 1155.958,A -85,B 0,C 180,E1 25996.118,E2 25996.118} C_VEL
LIN {X 0,Y 537.169,Z 1148.944,A -85,B 0,C 180,E1 25993.787,E2 25993.787} C_VEL
LIN {X 0,Y 538.087,Z 1140.028,A -85,B 0,C 180,E1 25991.249,E2 25991.249} C_VEL
LIN {X 0,Y 539.631,Z 1127.52,A -85,B 0,C 180,E1 25988.249,E2 25988.249} C_VEL
LIN {X 0,Y 541.244,Z 1116.211,A -85,B 0,C 180,E1 25985.904,E2 25985.904} C_VEL
LIN {X 0,Y 543.174,Z 1104.059,A -85,B 0,C 180,E1 25983.665,E2 25983.665} C_VEL
LIN {X 0,Y 545.983,Z 1088.284,A -85,B 0,C 180,E1 25981.088,E2 25981.088} C_VEL
LIN {X 0,Y 549.011,Z 1071.671,A -85,B 0,C 180,E1 25978.732,E2 25978.732} C_VEL
LIN {X 0,Y 551.913,Z 1056.655,A -85,B 0,C 180,E1 25976.825,E2 25976.825} C_VEL
LIN {X 0,Y 555.759,Z 1037.698,A -85,B 0,C 180,E1 25974.662,E2 25974.662} C_VEL
LIN {X 0,Y 560.026,Z 1016.697,A -85,B 0,C 180,E1 25972.561,E2 25972.561} C_VEL
LIN {X 0,Y 563.633,Z 998.644,A -85,B 0,C 180,E1 25970.968,E2 25970.968} C_VEL
LIN {X 0,Y 566.983,Z 981.443,A -85,B 0,C 180,E1 25969.61,E2 25969.61} C_VEL
LIN {X 0,Y 570.304,Z 963.734,A -85,B 0,C 180,E1 25968.359,E2 25968.359} C_VEL
LIN {X 0,Y 573.809,Z 944.018,A -85,B 0,C 180,E1 25967.122,E2 25967.122} C_VEL
LIN {X 0,Y 578.019,Z 918.433,A -85,B 0,C 180,E1 25965.739,E2 25965.739} C_VEL
LIN {X 0,Y 581.233,Z 896.054,A -85,B 0,C 180,E1 25964.717,E2 25964.717} C_VEL
LIN {X 0,Y 583.858,Z 876.017,A -85,B 0,C 180,E1 25963.937,E2 25963.937} C_VEL
LIN {X 0,Y 586.243,Z 855.095,A -85,B 0,C 180,E1 25963.246,E2 25963.246} C_VEL
LIN {X 0,Y 588.355,Z 833.377,A -85,B 0,C 180,E1 25962.656,E2 25962.656} C_VEL
LIN {X 0,Y 590.462,Z 806.358,A -85,B 0,C 180,E1 25962.087,E2 25962.087} C_VEL
LIN {X 0,Y 592.272,Z 761.512,A -85,B 0,C 180,E1 25961.416,E2 25961.416} C_VEL
LIN {X 0,Y 600.01,Z 538.759,A -85,B 0,C 180,E1 25958.19,E2 25958.19} C_VEL
LIN {X 0,Y 604.203,Z 421.597,A -85,B 0,C 180,E1 25956.449,E2 25956.449} C_VEL
LIN {X 0,Y 591.806,Z 404.256,A -85,B 0,C 180,E1 25954.413,E2 25954.413} C_VEL
LIN {X 0,Y 580.459,Z 389.424,A -85,B 0,C 180,E1 25952.393,E2 25952.393} C_VEL
LIN {X 0,Y 572.288,Z 379.12,A -85,B 0,C 180,E1 25950.821,E2 25950.821} C_VEL
LIN {X 0,Y 567.069,Z 372.789,A -85,B 0,C 180,E1 25949.759,E2 25949.759} C_VEL
LIN {X 0,Y 562.986,Z 367.756,A -85,B 0,C 180,E1 25948.887,E2 25948.887} C_VEL
LIN {X 0,Y 559.331,Z 363.225,A -85,B 0,C 180,E1 25948.073,E2 25948.073} C_VEL
LIN {X 0,Y 554.91,Z 358.446,A -85,B 0,C 180,E1 25947.064,E2 25947.064} C_VEL
LIN {X 0,Y 553.357,Z 356.236,A -85,B 0,C 180,E1 25946.681,E2 25946.681} C_VEL
LIN {X 0,Y 550.081,Z 353.055,A -85,B 0,C 180,E1 25945.894,E2 25945.894} C_VEL
LIN {X 0,Y 548.155,Z 350.085,A -85,B 0,C 180,E1 25945.383,E2 25945.383} C_VEL
LIN {X 0,Y 544.811,Z 347.217,A -85,B 0,C 180,E1 25944.534,E2 25944.534} C_VEL
LIN {X 0,Y 543.044,Z 343.876,A -85,B 0,C 180,E1 25944.012,E2 25944.012} C_VEL
LIN {X 0,Y 539.889,Z 341.932,A -85,B 0,C 180,E1 25943.176,E2 25943.176} C_VEL
LIN {X 0,Y 538.069,Z 339.266,A -85,B 0,C 180,E1 25942.623,E2 25942.623} C_VEL
LIN {X 0,Y 537.538,Z 337.256,A -85,B 0,C 180,E1 25942.414,E2 25942.414} C_VEL
LIN {X 0,Y 537.595,Z 337.218,A -85,B 0,C 180,E1 25939.221,E2 25939.221} C_VEL
LIN {X 0,Y 537.537,Z 337.226,A -85,B 0,C 180,E1 25935.98,E2 25935.98} C_VEL
LIN {X 0,Y 537.6,Z 337.242,A -85,B 0,C 180,E1 25932.787,E2 25932.787} C_VEL
LIN {X 0,Y 537.547,Z 337.214,A -85,B 0,C 180,E1 25929.637,E2 25929.637} C_VEL
LIN {X 0,Y 537.565,Z 337.268,A -85,B 0,C 180,E1 25926.193,E2 25926.193} C_VEL
LIN {X 0,Y 537.594,Z 337.201,A -85,B 0,C 180,E1 25922.985,E2 25922.985} C_VEL
LIN {X 0,Y 537.559,Z 337.27,A -85,B 0,C 180,E1 25919.68,E2 25919.68} C_VEL
LIN {X 0,Y 537.603,Z 337.201,A -85,B 0,C 180,E1 25916.374,E2 25916.374} C_VEL
LIN {X 0,Y 537.576,Z 337.26,A -85,B 0,C 180,E1 25913.163,E2 25913.163} C_VEL
LIN {X 0,Y 537.571,Z 337.216,A -85,B 0,C 180,E1 25909.709,E2 25909.709} C_VEL
LIN {X 0,Y 537.625,Z 337.221,A -85,B 0,C 180,E1 25906.447,E2 25906.447} C_VEL
LIN {X 0,Y 537.577,Z 337.245,A -85,B 0,C 180,E1 25903.132,E2 25903.132} C_VEL
LIN {X 0,Y 537.599,Z 337.207,A -85,B 0,C 180,E1 25899.76,E2 25899.76} C_VEL
LIN {X 0,Y 537.613,Z 337.333,A -85,B 0,C 180,E1 25898.678,E2 25898.678} C_VEL
LIN {X 0,Y 539.128,Z 341.048,A -85,B 0,C 180,E1 25897.654,E2 25897.654} C_VEL
LIN {X 0,Y 540.792,Z 343.034,A -85,B 0,C 180,E1 25896.98,E2 25896.98} C_VEL
LIN {X 0,Y 543.742,Z 347.112,A -85,B 0,C 180,E1 25896.136,E2 25896.136} C_VEL
LIN {X 0,Y 546.049,Z 349.548,A -85,B 0,C 180,E1 25895.525,E2 25895.525} C_VEL
LIN {X 0,Y 549.893,Z 354.194,A -85,B 0,C 180,E1 25894.53,E2 25894.53} C_VEL
LIN {X 0,Y 555.737,Z 361.682,A -85,B 0,C 180,E1 25893.095,E2 25893.095} C_VEL
LIN {X 0,Y 559.912,Z 366.931,A -85,B 0,C 180,E1 25892.132,E2 25892.132} C_VEL
LIN {X 0,Y 565.385,Z 374.023,A -85,B 0,C 180,E1 25890.928,E2 25890.928} C_VEL
LIN {X 0,Y 572.058,Z 382.905,A -85,B 0,C 180,E1 25889.543,E2 25889.543} C_VEL
LIN {X 0,Y 581.799,Z 396.228,A -85,B 0,C 180,E1 25887.661,E2 25887.661} C_VEL
LIN {X 0,Y 593.848,Z 413.738,A -85,B 0,C 180,E1 25885.517,E2 25885.517} C_VEL
LIN {X 0,Y 604.517,Z 430.257,A -85,B 0,C 180,E1 25883.757,E2 25883.757} C_VEL
LIN {X 0,Y 596.805,Z 645.056,A -85,B 0,C 180,E1 25880.614,E2 25880.614} C_VEL
LIN {X 0,Y 590.598,Z 824.815,A -85,B 0,C 180,E1 25878.013,E2 25878.013} C_VEL
LIN {X 0,Y 588.932,Z 849.528,A -85,B 0,C 180,E1 25877.56,E2 25877.56} C_VEL
LIN {X 0,Y 586.299,Z 877.877,A -85,B 0,C 180,E1 25876.85,E2 25876.85} C_VEL
LIN {X 0,Y 583.768,Z 900.178,A -85,B 0,C 180,E1 25876.143,E2 25876.143} C_VEL
LIN {X 0,Y 581.102,Z 920.987,A -85,B 0,C 180,E1 25875.355,E2 25875.355} C_VEL
LIN {X 0,Y 578.215,Z 941.397,A -85,B 0,C 180,E1 25874.453,E2 25874.453} C_VEL
LIN {X 0,Y 574.349,Z 966.466,A -85,B 0,C 180,E1 25873.169,E2 25873.169} C_VEL
LIN {X 0,Y 570.367,Z 989.528,A -85,B 0,C 180,E1 25871.77,E2 25871.77} C_VEL
LIN {X 0,Y 566.941,Z 1008.476,A -85,B 0,C 180,E1 25870.467,E2 25870.467} C_VEL
LIN {X 0,Y 563.615,Z 1026.253,A -85,B 0,C 180,E1 25869.099,E2 25869.099} C_VEL
LIN {X 0,Y 560.246,Z 1043.889,A -85,B 0,C 180,E1 25867.587,E2 25867.587} C_VEL
LIN {X 0,Y 556.527,Z 1063.326,A -85,B 0,C 180,E1 25865.725,E2 25865.725} C_VEL
LIN {X 0,Y 552.54,Z 1083.588,A -85,B 0,C 180,E1 25863.499,E2 25863.499} C_VEL
LIN {X 0,Y 549.553,Z 1098.823,A -85,B 0,C 180,E1 25861.6,E2 25861.6} C_VEL
LIN {X 0,Y 546.948,Z 1112.602,A -85,B 0,C 180,E1 25859.696,E2 25859.696} C_VEL
LIN {X 0,Y 544.607,Z 1125.772,A -85,B 0,C 180,E1 25857.677,E2 25857.677} C_VEL
LIN {X 0,Y 542.107,Z 1140.844,A -85,B 0,C 180,E1 25855.092,E2 25855.092} C_VEL
LIN {X 0,Y 540.077,Z 1154.229,A -85,B 0,C 180,E1 25852.419,E2 25852.419} C_VEL
LIN {X 0,Y 538.721,Z 1164.521,A -85,B 0,C 180,E1 25850.081,E2 25850.081} C_VEL
LIN {X 0,Y 537.703,Z 1173.512,A -85,B 0,C 180,E1 25847.756,E2 25847.756} C_VEL
LIN {X 0,Y 536.844,Z 1183.174,A -85,B 0,C 180,E1 25844.837,E2 25844.837} C_VEL
LIN {X 0,Y 536.324,Z 1190.568,A -85,B 0,C 180,E1 25842.052,E2 25842.052} C_VEL
LIN {X 0,Y 536.091,Z 1195.702,A -85,B 0,C 180,E1 25839.663,E2 25839.663} C_VEL
LIN {X 0,Y 535.978,Z 1199.686,A -85,B 0,C 180,E1 25837.288,E2 25837.288} C_VEL
LIN {X 0,Y 535.918,Z 1202.89,A -85,B 0,C 180,E1 25834.601,E2 25834.601} C_VEL
LIN {X 0,Y 535.908,Z 1204.645,A -85,B 0,C 180,E1 25831.711,E2 25831.711} C_VEL
LIN {X 0,Y 535.899,Z 1204.849,A -85,B 0,C 180,E1 25829.252,E2 25829.252} C_VEL
LIN {X 0,Y 535.916,Z 1203.972,A -85,B 0,C 180,E1 25826.898,E2 25826.898} C_VEL
LIN {X 0,Y 535.932,Z 1201.98,A -85,B 0,C 180,E1 25824.54,E2 25824.54} C_VEL
LIN {X 0,Y 535.999,Z 1198.727,A -85,B 0,C 180,E1 25822.066,E2 25822.066} C_VEL
LIN {X 0,Y 536.184,Z 1193.351,A -85,B 0,C 180,E1 25819.144,E2 25819.144} C_VEL
LIN {X 0,Y 536.58,Z 1186.672,A -85,B 0,C 180,E1 25816.421,E2 25816.421} C_VEL
LIN {X 0,Y 537.085,Z 1179.858,A -85,B 0,C 180,E1 25814.118,E2 25814.118} C_VEL
LIN {X 0,Y 537.886,Z 1171.844,A -85,B 0,C 180,E1 25811.79,E2 25811.79} C_VEL
LIN {X 0,Y 539.073,Z 1161.773,A -85,B 0,C 180,E1 25809.252,E2 25809.252} C_VEL
LIN {X 0,Y 540.935,Z 1148.287,A -85,B 0,C 180,E1 25806.353,E2 25806.353} C_VEL
LIN {X 0,Y 542.817,Z 1136.36,A -85,B 0,C 180,E1 25804.116,E2 25804.116} C_VEL
LIN {X 0,Y 545.002,Z 1123.401,A -85,B 0,C 180,E1 25801.942,E2 25801.942} C_VEL
LIN {X 0,Y 548.028,Z 1107.206,A -85,B 0,C 180,E1 25799.522,E2 25799.522} C_VEL
LIN {X 0,Y 551.436,Z 1089.143,A -85,B 0,C 180,E1 25797.17,E2 25797.17} C_VEL
LIN {X 0,Y 554.455,Z 1073.791,A -85,B 0,C 180,E1 25795.386,E2 25795.386} C_VEL
LIN {X 0,Y 557.663,Z 1057.135,A -85,B 0,C 180,E1 25793.661,E2 25793.661} C_VEL
LIN {X 0,Y 561.235,Z 1038.685,A -85,B 0,C 180,E1 25791.946,E2 25791.946} C_VEL
LIN {X 0,Y 565.855,Z 1014.408,A -85,B 0,C 180,E1 25789.971,E2 25789.971} C_VEL
LIN {X 0,Y 569.482,Z 994.438,A -85,B 0,C 180,E1 25788.554,E2 25788.554} C_VEL
LIN {X 0,Y 572.754,Z 975.567,A -85,B 0,C 180,E1 25787.365,E2 25787.365} C_VEL
LIN {X 0,Y 575.994,Z 955.696,A -85,B 0,C 180,E1 25786.256,E2 25786.256} C_VEL
LIN {X 0,Y 579.567,Z 932.293,A -85,B 0,C 180,E1 25785.122,E2 25785.122} C_VEL
LIN {X 0,Y 583.15,Z 905.388,A -85,B 0,C 180,E1 25784.042,E2 25784.042} C_VEL
LIN {X 0,Y 585.694,Z 883.419,A -85,B 0,C 180,E1 25783.314,E2 25783.314} C_VEL
LIN {X 0,Y 587.812,Z 862.127,A -85,B 0,C 180,E1 25782.732,E2 25782.732} C_VEL
LIN {X 0,Y 589.621,Z 840.235,A -85,B 0,C 180,E1 25782.256,E2 25782.256} C_VEL
LIN {X 0,Y 591.202,Z 812.264,A -85,B 0,C 180,E1 25781.792,E2 25781.792} C_VEL
LIN {X 0,Y 598.778,Z 588.155,A -85,B 0,C 180,E1 25778.561,E2 25778.561} C_VEL
LIN {X 0,Y 604.407,Z 430.078,A -85,B 0,C 180,E1 25776.229,E2 25776.229} C_VEL
LIN {X 0,Y 591.605,Z 410.39,A -85,B 0,C 180,E1 25774.105,E2 25774.105} C_VEL
LIN {X 0,Y 578.502,Z 391.542,A -85,B 0,C 180,E1 25771.727,E2 25771.727} C_VEL
LIN {X 0,Y 567.062,Z 376.108,A -85,B 0,C 180,E1 25769.44,E2 25769.44} C_VEL
LIN {X 0,Y 561.918,Z 369.604,A -85,B 0,C 180,E1 25768.337,E2 25768.337} C_VEL
LIN {X 0,Y 557.992,Z 364.491,A -85,B 0,C 180,E1 25767.45,E2 25767.45} C_VEL
LIN {X 0,Y 553.083,Z 358.332,A -85,B 0,C 180,E1 25766.291,E2 25766.291} C_VEL
LIN {X 0,Y 549.217,Z 353.56,A -85,B 0,C 180,E1 25765.33,E2 25765.33} C_VEL
LIN {X 0,Y 544.759,Z 348.067,A -85,B 0,C 180,E1 25764.162,E2 25764.162} C_VEL
LIN {X 0,Y 541.355,Z 344.047,A -85,B 0,C 180,E1 25763.225,E2 25763.225} C_VEL
LIN {X 0,Y 540.559,Z 342.547,A -85,B 0,C 180,E1 25762.973,E2 25762.973} C_VEL
LIN {X 0,Y 538.294,Z 339.578,A -85,B 0,C 180,E1 25761.923,E2 25761.923} C_VEL
LIN {X 0,Y 537.596,Z 337.219,A -85,B 0,C 180,E1 25761.265,E2 25761.265} C_VEL
LIN {X 0,Y 537.625,Z 337.259,A -85,B 0,C 180,E1 25757.871,E2 25757.871} C_VEL
LIN {X 0,Y 537.569,Z 337.209,A -85,B 0,C 180,E1 25754.543,E2 25754.543} C_VEL
LIN {X 0,Y 537.601,Z 337.246,A -85,B 0,C 180,E1 25751.153,E2 25751.153} C_VEL
LIN {X 0,Y 537.606,Z 337.219,A -85,B 0,C 180,E1 25747.803,E2 25747.803} C_VEL
LIN {X 0,Y 537.563,Z 337.225,A -85,B 0,C 180,E1 25744.478,E2 25744.478} C_VEL
LIN {X 0,Y 537.618,Z 337.237,A -85,B 0,C 180,E1 25741.172,E2 25741.172} C_VEL
LIN {X 0,Y 537.558,Z 337.218,A -85,B 0,C 180,E1 25738.081,E2 25738.081} C_VEL
LIN {X 0,Y 537.576,Z 337.256,A -85,B 0,C 180,E1 25734.664,E2 25734.664} C_VEL
LIN {X 0,Y 537.566,Z 337.211,A -85,B 0,C 180,E1 25731.658,E2 25731.658} C_VEL
LIN {X 0,Y 537.558,Z 337.269,A -85,B 0,C 180,E1 25728.302,E2 25728.302} C_VEL
LIN {X 0,Y 537.617,Z 337.201,A -85,B 0,C 180,E1 25725.018,E2 25725.018} C_VEL
LIN {X 0,Y 537.548,Z 337.264,A -85,B 0,C 180,E1 25721.79,E2 25721.79} C_VEL
LIN {X 0,Y 537.569,Z 337.221,A -85,B 0,C 180,E1 25718.431,E2 25718.431} C_VEL
LIN {X 0,Y 537.572,Z 337.409,A -85,B 0,C 180,E1 25717.443,E2 25717.443} C_VEL
LIN {X 0,Y 538.51,Z 340.137,A -85,B 0,C 180,E1 25717.108,E2 25717.108} C_VEL
LIN {X 0,Y 541.123,Z 342.958,A -85,B 0,C 180,E1 25716.361,E2 25716.361} C_VEL
LIN {X 0,Y 543.146,Z 344.14,A -85,B 0,C 180,E1 25715.834,E2 25715.834} C_VEL
LIN {X 0,Y 545.164,Z 347.639,A -85,B 0,C 180,E1 25715.251,E2 25715.251} C_VEL
LIN {X 0,Y 548.631,Z 350.574,A -85,B 0,C 180,E1 25714.38,E2 25714.38} C_VEL
LIN {X 0,Y 551.239,Z 354.444,A -85,B 0,C 180,E1 25713.702,E2 25713.702} C_VEL
LIN {X 0,Y 553.968,Z 356.888,A -85,B 0,C 180,E1 25713.061,E2 25713.061} C_VEL
LIN {X 0,Y 557.143,Z 361.153,A -85,B 0,C 180,E1 25712.301,E2 25712.301} C_VEL
LIN {X 0,Y 559.351,Z 363.283,A -85,B 0,C 180,E1 25711.812,E2 25711.812} C_VEL
LIN {X 0,Y 563.018,Z 367.793,A -85,B 0,C 180,E1 25710.998,E2 25710.998} C_VEL
LIN {X 0,Y 569.314,Z 375.515,A -85,B 0,C 180,E1 25709.673,E2 25709.673} C_VEL
LIN {X 0,Y 577.495,Z 385.566,A -85,B 0,C 180,E1 25708.065,E2 25708.065} C_VEL
LIN {X 0,Y 587.336,Z 398.48,A -85,B 0,C 180,E1 25706.261,E2 25706.261} C_VEL
LIN {X 0,Y 597.522,Z 412.141,A -85,B 0,C 180,E1 25704.532,E2 25704.532} C_VEL
LIN {X 0,Y 604.307,Z 422.052,A -85,B 0,C 180,E1 25703.435,E2 25703.435} C_VEL
LIN {X 0,Y 596.473,Z 637.953,A -85,B 0,C 180,E1 25700.275,E2 25700.275} C_VEL
LIN {X 0,Y 590.823,Z 798.976,A -85,B 0,C 180,E1 25697.941,E2 25697.941} C_VEL
LIN {X 0,Y 590.315,Z 808.486,A -85,B 0,C 180,E1 25697.784,E2 25697.784} C_VEL
LIN {X 0,Y 589.022,Z 816.105,A -85,B 0,C 180,E1 25697.716,E2 25697.716} C_VEL
LIN {X 0,Y 583.928,Z 833.256,A -85,B 0,C 180,E1 25697.743,E2 25697.743} C_VEL
LIN {X 0,Y 582.195,Z 841.871,A -85,B 0,C 180,E1 25697.624,E2 25697.624} C_VEL
LIN {X 0,Y 582.086,Z 842.944,A -85,B 0,C 180,E1 25697.598,E2 25697.598} C_VEL
LIN {X 0,Y 579.076,Z 870.011,A -85,B 0,C 180,E1 25696.773,E2 25696.773} C_VEL
LIN {X 0,Y 576.125,Z 892.347,A -85,B 0,C 180,E1 25695.93,E2 25695.93} C_VEL
LIN {X 0,Y 573.183,Z 912.262,A -85,B 0,C 180,E1 25695.049,E2 25695.049} C_VEL
LIN {X 0,Y 569.847,Z 932.618,A -85,B 0,C 180,E1 25694.013,E2 25694.013} C_VEL
LIN {X 0,Y 565.662,Z 956.485,A -85,B 0,C 180,E1 25692.608,E2 25692.608} C_VEL
LIN {X 0,Y 561.23,Z 979.199,A -85,B 0,C 180,E1 25691.033,E2 25691.033} C_VEL
LIN {X 0,Y 557.542,Z 997.347,A -85,B 0,C 180,E1 25689.608,E2 25689.608} C_VEL
LIN {X 0,Y 553.932,Z 1014.587,A -85,B 0,C 180,E1 25688.092,E2 25688.092} C_VEL
LIN {X 0,Y 550.157,Z 1032.461,A -85,B 0,C 180,E1 25686.333,E2 25686.333} C_VEL
LIN {X 0,Y 545.562,Z 1053.88,A -85,B 0,C 180,E1 25683.922,E2 25683.922} C_VEL
LIN {X 0,Y 541.956,Z 1071.051,A -85,B 0,C 180,E1 25681.722,E2 25681.722} C_VEL
LIN {X 0,Y 538.878,Z 1086.938,A -85,B 0,C 180,E1 25679.452,E2 25679.452} C_VEL
LIN {X 0,Y 535.757,Z 1103.578,A -85,B 0,C 180,E1 25676.729,E2 25676.729} C_VEL
LIN {X 0,Y 533.659,Z 1116.008,A -85,B 0,C 180,E1 25674.412,E2 25674.412} C_VEL
LIN {X 0,Y 531.954,Z 1127.137,A -85,B 0,C 180,E1 25672.078,E2 25672.078} C_VEL
LIN {X 0,Y 530.344,Z 1139.294,A -85,B 0,C 180,E1 25669.15,E2 25669.15} C_VEL
LIN {X 0,Y 529.308,Z 1148.657,A -85,B 0,C 180,E1 25666.46,E2 25666.46} C_VEL
LIN {X 0,Y 528.698,Z 1155.638,A -85,B 0,C 180,E1 25664.12,E2 25664.12} C_VEL
LIN {X 0,Y 528.295,Z 1161.733,A -85,B 0,C 180,E1 25661.684,E2 25661.684} C_VEL
LIN {X 0,Y 528.052,Z 1167.266,A -85,B 0,C 180,E1 25658.932,E2 25658.932} C_VEL
LIN {X 0,Y 527.945,Z 1171.476,A -85,B 0,C 180,E1 25655.979,E2 25655.979} C_VEL
LIN {X 0,Y 527.915,Z 1173.738,A -85,B 0,C 180,E1 25653.473,E2 25653.473} C_VEL
LIN {X 0,Y 527.911,Z 1174.749,A -85,B 0,C 180,E1 25651.194,E2 25651.194} C_VEL
LIN {X 0,Y 527.906,Z 1174.813,A -85,B 0,C 180,E1 25649.023,E2 25649.023} C_VEL
LIN {X 0,Y 527.912,Z 1173.93,A -85,B 0,C 180,E1 25646.743,E2 25646.743} C_VEL
LIN {X 0,Y 527.933,Z 1171.912,A -85,B 0,C 180,E1 25644.348,E2 25644.348} C_VEL
LIN {X 0,Y 528.018,Z 1168.471,A -85,B 0,C 180,E1 25641.726,E2 25641.726} C_VEL
LIN {X 0,Y 528.236,Z 1162.703,A -85,B 0,C 180,E1 25638.647,E2 25638.647} C_VEL
LIN {X 0,Y 528.637,Z 1156.489,A -85,B 0,C 180,E1 25636.101,E2 25636.101} C_VEL
LIN {X 0,Y 529.199,Z 1149.647,A -85,B 0,C 180,E1 25633.762,E2 25633.762} C_VEL
LIN {X 0,Y 530.05,Z 1141.645,A -85,B 0,C 180,E1 25631.41,E2 25631.41} C_VEL
LIN {X 0,Y 531.414,Z 1131.021,A -85,B 0,C 180,E1 25628.708,E2 25628.708} C_VEL
LIN {X 0,Y 533.345,Z 1117.925,A -85,B 0,C 180,E1 25625.878,E2 25625.878} C_VEL
LIN {X 0,Y 535.336,Z 1105.958,A -85,B 0,C 180,E1 25623.608,E2 25623.608} C_VEL
LIN {X 0,Y 537.633,Z 1093.228,A -85,B 0,C 180,E1 25621.448,E2 25621.448} C_VEL
LIN {X 0,Y 540.902,Z 1076.712,A -85,B 0,C 180,E1 25618.954,E2 25618.954} C_VEL
LIN {X 0,Y 544.756,Z 1057.551,A -85,B 0,C 180,E1 25616.441,E2 25616.441} C_VEL
LIN {X 0,Y 548.009,Z 1042.324,A -85,B 0,C 180,E1 25614.646,E2 25614.646} C_VEL
LIN {X 0,Y 551.732,Z 1025.01,A -85,B 0,C 180,E1 25612.816,E2 25612.816} C_VEL
LIN {X 0,Y 556.577,Z 1002.207,A -85,B 0,C 180,E1 25610.71,E2 25610.71} C_VEL
LIN {X 0,Y 560.319,Z 983.812,A -85,B 0,C 180,E1 25609.224,E2 25609.224} C_VEL
LIN {X 0,Y 563.72,Z 966.484,A -85,B 0,C 180,E1 25607.974,E2 25607.974} C_VEL
LIN {X 0,Y 567.183,Z 947.845,A -85,B 0,C 180,E1 25606.775,E2 25606.775} C_VEL
LIN {X 0,Y 570.644,Z 927.916,A -85,B 0,C 180,E1 25605.645,E2 25605.645} C_VEL
LIN {X 0,Y 574.678,Z 902.887,A -85,B 0,C 180,E1 25604.422,E2 25604.422} C_VEL
LIN {X 0,Y 578.011,Z 878.475,A -85,B 0,C 180,E1 25603.44,E2 25603.44} C_VEL
LIN {X 0,Y 580.589,Z 856.864,A -85,B 0,C 180,E1 25602.713,E2 25602.713} C_VEL
LIN {X 0,Y 582.738,Z 835.842,A -85,B 0,C 180,E1 25602.132,E2 25602.132} C_VEL
LIN {X 0,Y 584.552,Z 813.957,A -85,B 0,C 180,E1 25601.647,E2 25601.647} C_VEL
LIN {X 0,Y 586.184,Z 785.231,A -85,B 0,C 180,E1 25601.168,E2 25601.168} C_VEL
LIN {X 0,Y 594.253,Z 561.291,A -85,B 0,C 180,E1 25597.912,E2 25597.912} C_VEL
LIN {X 0,Y 599.373,Z 425.888,A -85,B 0,C 180,E1 25595.901,E2 25595.901} C_VEL
LIN {X 0,Y 586.051,Z 407.339,A -85,B 0,C 180,E1 25593.644,E2 25593.644} C_VEL
LIN {X 0,Y 576.57,Z 395.026,A -85,B 0,C 180,E1 25591.904,E2 25591.904} C_VEL
LIN {X 0,Y 569.418,Z 385.902,A -85,B 0,C 180,E1 25590.496,E2 25590.496} C_VEL
LIN {X 0,Y 564.26,Z 379.575,A -85,B 0,C 180,E1 25589.426,E2 25589.426} C_VEL
LIN {X 0,Y 560.221,Z 374.6,A -85,B 0,C 180,E1 25588.547,E2 25588.547} C_VEL
LIN {X 0,Y 555.99,Z 369.44,A -85,B 0,C 180,E1 25587.587,E2 25587.587} C_VEL
LIN {X 0,Y 552.36,Z 365.325,A -85,B 0,C 180,E1 25586.733,E2 25586.733} C_VEL
LIN {X 0,Y 551.007,Z 363.496,A -85,B 0,C 180,E1 25586.397,E2 25586.397} C_VEL
LIN {X 0,Y 547.504,Z 359.804,A -85,B 0,C 180,E1 25585.531,E2 25585.531} C_VEL
LIN {X 0,Y 545.86,Z 357.421,A -85,B 0,C 180,E1 25585.091,E2 25585.091} C_VEL
LIN {X 0,Y 542.491,Z 354.239,A -85,B 0,C 180,E1 25584.211,E2 25584.211} C_VEL
LIN {X 0,Y 540.608,Z 351.297,A -85,B 0,C 180,E1 25583.663,E2 25583.663} C_VEL
LIN {X 0,Y 537.294,Z 348.641,A -85,B 0,C 180,E1 25582.744,E2 25582.744} C_VEL
LIN {X 0,Y 535.412,Z 345.301,A -85,B 0,C 180,E1 25582.137,E2 25582.137} C_VEL
LIN {X 0,Y 534.813,Z 344.762,A -85,B 0,C 180,E1 25581.958,E2 25581.958} C_VEL
LIN {X 0,Y 531.78,Z 342.703,A -85,B 0,C 180,E1 25581.047,E2 25581.047} C_VEL
LIN {X 0,Y 530.066,Z 340.065,A -85,B 0,C 180,E1 25580.454,E2 25580.454} C_VEL
LIN {X 0,Y 529.594,Z 338.2,A -85,B 0,C 180,E1 25580.213,E2 25580.213} C_VEL
LIN {X 0,Y 529.658,Z 338.236,A -85,B 0,C 180,E1 25576.901,E2 25576.901} C_VEL
LIN {X 0,Y 529.603,Z 338.206,A -85,B 0,C 180,E1 25573.762,E2 25573.762} C_VEL
LIN {X 0,Y 529.62,Z 338.215,A -85,B 0,C 180,E1 25570.332,E2 25570.332} C_VEL
LIN {X 0,Y 529.659,Z 338.22,A -85,B 0,C 180,E1 25567.048,E2 25567.048} C_VEL
LIN {X 0,Y 529.61,Z 338.204,A -85,B 0,C 180,E1 25563.789,E2 25563.789} C_VEL
LIN {X 0,Y 529.667,Z 338.239,A -85,B 0,C 180,E1 25560.433,E2 25560.433} C_VEL
LIN {X 0,Y 529.631,Z 338.194,A -85,B 0,C 180,E1 25557.186,E2 25557.186} C_VEL
LIN {X 0,Y 529.631,Z 338.257,A -85,B 0,C 180,E1 25553.714,E2 25553.714} C_VEL
LIN {X 0,Y 529.68,Z 338.187,A -85,B 0,C 180,E1 25550.438,E2 25550.438} C_VEL
LIN {X 0,Y 529.637,Z 338.237,A -85,B 0,C 180,E1 25547.128,E2 25547.128} C_VEL
LIN {X 0,Y 529.644,Z 338.213,A -85,B 0,C 180,E1 25543.663,E2 25543.663} C_VEL
LIN {X 0,Y 529.679,Z 338.341,A -85,B 0,C 180,E1 25540.652,E2 25540.652} C_VEL
LIN {X 0,Y 531.346,Z 342.22,A -85,B 0,C 180,E1 25539.512,E2 25539.512} C_VEL
LIN {X 0,Y 533.766,Z 344.631,A -85,B 0,C 180,E1 25538.747,E2 25538.747} C_VEL
LIN {X 0,Y 537.031,Z 348.802,A -85,B 0,C 180,E1 25537.735,E2 25537.735} C_VEL
LIN {X 0,Y 538.768,Z 350.516,A -85,B 0,C 180,E1 25537.235,E2 25537.235} C_VEL
LIN {X 0,Y 542.06,Z 354.84,A -85,B 0,C 180,E1 25536.289,E2 25536.289} C_VEL
LIN {X 0,Y 544.244,Z 357.315,A -85,B 0,C 180,E1 25535.699,E2 25535.699} C_VEL
LIN {X 0,Y 549.084,Z 363.455,A -85,B 0,C 180,E1 25534.432,E2 25534.432} C_VEL
LIN {X 0,Y 553.365,Z 368.837,A -85,B 0,C 180,E1 25533.377,E2 25533.377} C_VEL
LIN {X 0,Y 557.593,Z 374.254,A -85,B 0,C 180,E1 25532.383,E2 25532.383} C_VEL
LIN {X 0,Y 562.911,Z 381.185,A -85,B 0,C 180,E1 25531.196,E2 25531.196} C_VEL
LIN {X 0,Y 569.407,Z 389.949,A -85,B 0,C 180,E1 25529.824,E2 25529.824} C_VEL
LIN {X 0,Y 578.937,Z 403.148,A -85,B 0,C 180,E1 25527.95,E2 25527.95} C_VEL
LIN {X 0,Y 590.629,Z 420.326,A -85,B 0,C 180,E1 25525.831,E2 25525.831} C_VEL
LIN {X 0,Y 599.612,Z 434.392,A -85,B 0,C 180,E1 25524.314,E2 25524.314} C_VEL
LIN {X 0,Y 591.565,Z 649.185,A -85,B 0,C 180,E1 25521.153,E2 25521.153} C_VEL
LIN {X 0,Y 585.241,Z 824.593,A -85,B 0,C 180,E1 25518.598,E2 25518.598} C_VEL
LIN {X 0,Y 583.493,Z 849.598,A -85,B 0,C 180,E1 25518.138,E2 25518.138} C_VEL
LIN {X 0,Y 580.762,Z 877.783,A -85,B 0,C 180,E1 25517.429,E2 25517.429} C_VEL
LIN {X 0,Y 578.155,Z 899.915,A -85,B 0,C 180,E1 25516.725,E2 25516.725} C_VEL
LIN {X 0,Y 575.402,Z 920.591,A -85,B 0,C 180,E1 25515.94,E2 25515.94} C_VEL
LIN {X 0,Y 572.368,Z 941.127,A -85,B 0,C 180,E1 25515.031,E2 25515.031} C_VEL
LIN {X 0,Y 568.337,Z 966.194,A -85,B 0,C 180,E1 25513.74,E2 25513.74} C_VEL
LIN {X 0,Y 564.187,Z 989.254,A -85,B 0,C 180,E1 25512.333,E2 25512.333} C_VEL
LIN {X 0,Y 560.605,Z 1008.202,A -85,B 0,C 180,E1 25511.021,E2 25511.021} C_VEL
LIN {X 0,Y 556.995,Z 1026.653,A -85,B 0,C 180,E1 25509.587,E2 25509.587} C_VEL
LIN {X 0,Y 553.29,Z 1045.19,A -85,B 0,C 180,E1 25507.975,E2 25507.975} C_VEL
LIN {X 0,Y 548.819,Z 1067.344,A -85,B 0,C 180,E1 25505.789,E2 25505.789} C_VEL
LIN {X 0,Y 545.144,Z 1085.324,A -85,B 0,C 180,E1 25503.761,E2 25503.761} C_VEL
LIN {X 0,Y 542.424,Z 1098.822,A -85,B 0,C 180,E1 25502.064,E2 25502.064} C_VEL
LIN {X 0,Y 539.573,Z 1113.062,A -85,B 0,C 180,E1 25500.07,E2 25500.07} C_VEL
LIN {X 0,Y 537.05,Z 1126.47,A -85,B 0,C 180,E1 25497.98,E2 25497.98} C_VEL
LIN {X 0,Y 534.336,Z 1141.971,A -85,B 0,C 180,E1 25495.254,E2 25495.254} C_VEL
LIN {X 0,Y 532.295,Z 1154.742,A -85,B 0,C 180,E1 25492.648,E2 25492.648} C_VEL
LIN {X 0,Y 530.871,Z 1164.978,A -85,B 0,C 180,E1 25490.276,E2 25490.276} C_VEL
LIN {X 0,Y 529.754,Z 1174.321,A -85,B 0,C 180,E1 25487.804,E2 25487.804} C_VEL
LIN {X 0,Y 528.818,Z 1184.246,A -85,B 0,C 180,E1 25484.676,E2 25484.676} C_VEL
LIN {X 0,Y 528.341,Z 1190.819,A -85,B 0,C 180,E1 25482.126,E2 25482.126} C_VEL
LIN {X 0,Y 528.098,Z 1195.905,A -85,B 0,C 180,E1 25479.701,E2 25479.701} C_VEL
LIN {X 0,Y 527.973,Z 1200.003,A -85,B 0,C 180,E1 25477.18,E2 25477.18} C_VEL
LIN {X 0,Y 527.919,Z 1203.273,A -85,B 0,C 180,E1 25474.236,E2 25474.236} C_VEL
LIN {X 0,Y 527.909,Z 1204.69,A -85,B 0,C 180,E1 25471.519,E2 25471.519} C_VEL
LIN {X 0,Y 527.899,Z 1204.849,A -85,B 0,C 180,E1 25469.24,E2 25469.24} C_VEL
LIN {X 0,Y 527.916,Z 1203.969,A -85,B 0,C 180,E1 25466.851,E2 25466.851} C_VEL
LIN {X 0,Y 527.934,Z 1201.977,A -85,B 0,C 180,E1 25464.457,E2 25464.457} C_VEL
LIN {X 0,Y 528.006,Z 1198.724,A -85,B 0,C 180,E1 25461.945,E2 25461.945} C_VEL
LIN {X 0,Y 528.204,Z 1193.351,A -85,B 0,C 180,E1 25458.978,E2 25458.978} C_VEL
LIN {X 0,Y 528.632,Z 1186.669,A -85,B 0,C 180,E1 25456.213,E2 25456.213} C_VEL
LIN {X 0,Y 529.178,Z 1179.857,A -85,B 0,C 180,E1 25453.874,E2 25453.874} C_VEL
LIN {X 0,Y 530.029,Z 1171.89,A -85,B 0,C 180,E1 25451.523,E2 25451.523} C_VEL
LIN {X 0,Y 531.296,Z 1161.771,A -85,B 0,C 180,E1 25448.934,E2 25448.934} C_VEL
LIN {X 0,Y 533.287,Z 1148.285,A -85,B 0,C 180,E1 25445.993,E2 25445.993} C_VEL
LIN {X 0,Y 535.282,Z 1136.328,A -85,B 0,C 180,E1 25443.719,E2 25443.719} C_VEL
LIN {X 0,Y 537.55,Z 1123.669,A -85,B 0,C 180,E1 25441.565,E2 25441.565} C_VEL
LIN {X 0,Y 540.474,Z 1108.747,A -85,B 0,C 180,E1 25439.297,E2 25439.297} C_VEL
LIN {X 0,Y 544.202,Z 1090.024,A -85,B 0,C 180,E1 25436.804,E2 25436.804} C_VEL
LIN {X 0,Y 547.516,Z 1073.514,A -85,B 0,C 180,E1 25434.883,E2 25434.883} C_VEL
LIN {X 0,Y 550.805,Z 1057.29,A -85,B 0,C 180,E1 25433.184,E2 25433.184} C_VEL
LIN {X 0,Y 554.411,Z 1039.527,A -85,B 0,C 180,E1 25431.511,E2 25431.511} C_VEL
LIN {X 0,Y 559.069,Z 1016.361,A -85,B 0,C 180,E1 25429.586,E2 25429.586} C_VEL
LIN {X 0,Y 563.108,Z 995.066,A -85,B 0,C 180,E1 25428.054,E2 25428.054} C_VEL
LIN {X 0,Y 566.53,Z 976.203,A -85,B 0,C 180,E1 25426.852,E2 25426.852} C_VEL
LIN {X 0,Y 569.785,Z 957.095,A -85,B 0,C 180,E1 25425.771,E2 25425.771} C_VEL
LIN {X 0,Y 573.055,Z 936.577,A -85,B 0,C 180,E1 25424.755,E2 25424.755} C_VEL
LIN {X 0,Y 576.689,Z 911.669,A -85,B 0,C 180,E1 25423.698,E2 25423.698} C_VEL
LIN {X 0,Y 579.941,Z 885.083,A -85,B 0,C 180,E1 25422.788,E2 25422.788} C_VEL
LIN {X 0,Y 582.233,Z 863.139,A -85,B 0,C 180,E1 25422.179,E2 25422.179} C_VEL
LIN {X 0,Y 584.089,Z 841.753,A -85,B 0,C 180,E1 25421.706,E2 25421.706} C_VEL
LIN {X 0,Y 585.558,Z 818.311,A -85,B 0,C 180,E1 25421.303,E2 25421.303} C_VEL
LIN {X 0,Y 593.378,Z 598.844,A -85,B 0,C 180,E1 25418.113,E2 25418.113} C_VEL
LIN {X 0,Y 599.506,Z 434.166,A -85,B 0,C 180,E1 25415.672,E2 25415.672} C_VEL
LIN {X 0,Y 587.31,Z 415.407,A -85,B 0,C 180,E1 25413.595,E2 25413.595} C_VEL
LIN {X 0,Y 575.441,Z 398.135,A -85,B 0,C 180,E1 25411.389,E2 25411.389} C_VEL
LIN {X 0,Y 564.244,Z 382.87,A -85,B 0,C 180,E1 25409.107,E2 25409.107} C_VEL
LIN {X 0,Y 559.164,Z 376.368,A -85,B 0,C 180,E1 25407.995,E2 25407.995} C_VEL
LIN {X 0,Y 555.286,Z 371.289,A -85,B 0,C 180,E1 25407.102,E2 25407.102} C_VEL
LIN {X 0,Y 550.541,Z 365.268,A -85,B 0,C 180,E1 25405.958,E2 25405.958} C_VEL
LIN {X 0,Y 546.727,Z 360.525,A -85,B 0,C 180,E1 25404.991,E2 25404.991} C_VEL
LIN {X 0,Y 542.697,Z 355.447,A -85,B 0,C 180,E1 25403.912,E2 25403.912} C_VEL
LIN {X 0,Y 539.162,Z 351.194,A -85,B 0,C 180,E1 25402.92,E2 25402.92} C_VEL
LIN {X 0,Y 537.975,Z 349.601,A -85,B 0,C 180,E1 25402.57,E2 25402.57} C_VEL
LIN {X 0,Y 534.433,Z 345.733,A -85,B 0,C 180,E1 25401.513,E2 25401.513} C_VEL
LIN {X 0,Y 533.005,Z 343.777,A -85,B 0,C 180,E1 25401.054,E2 25401.054} C_VEL
LIN {X 0,Y 530.593,Z 341.059,A -85,B 0,C 180,E1 25400.173,E2 25400.173} C_VEL
LIN {X 0,Y 529.66,Z 338.202,A -85,B 0,C 180,E1 25399.289,E2 25399.289} C_VEL
LIN {X 0,Y 529.67,Z 338.204,A -85,B 0,C 180,E1 25395.999,E2 25395.999} C_VEL
LIN {X 0,Y 529.636,Z 338.242,A -85,B 0,C 180,E1 25392.65,E2 25392.65} C_VEL
LIN {X 0,Y 529.675,Z 338.188,A -85,B 0,C 180,E1 25389.343,E2 25389.343} C_VEL
LIN {X 0,Y 529.642,Z 338.258,A -85,B 0,C 180,E1 25386.069,E2 25386.069} C_VEL
LIN {X 0,Y 529.624,Z 338.195,A -85,B 0,C 180,E1 25382.597,E2 25382.597} C_VEL
LIN {X 0,Y 529.691,Z 338.238,A -85,B 0,C 180,E1 25379.351,E2 25379.351} C_VEL
LIN {X 0,Y 529.619,Z 338.203,A -85,B 0,C 180,E1 25375.994,E2 25375.994} C_VEL
LIN {X 0,Y 529.627,Z 338.217,A -85,B 0,C 180,E1 25372.515,E2 25372.515} C_VEL
LIN {X 0,Y 529.664,Z 338.217,A -85,B 0,C 180,E1 25369.229,E2 25369.229} C_VEL
LIN {X 0,Y 529.606,Z 338.206,A -85,B 0,C 180,E1 25366.015,E2 25366.015} C_VEL
LIN {X 0,Y 529.664,Z 338.243,A -85,B 0,C 180,E1 25362.759,E2 25362.759} C_VEL
LIN {X 0,Y 529.609,Z 338.243,A -85,B 0,C 180,E1 25359.615,E2 25359.615} C_VEL
LIN {X 0,Y 530.51,Z 340.981,A -85,B 0,C 180,E1 25359.247,E2 25359.247} C_VEL
LIN {X 0,Y 533.04,Z 343.816,A -85,B 0,C 180,E1 25358.428,E2 25358.428} C_VEL
LIN {X 0,Y 535.376,Z 345.173,A -85,B 0,C 180,E1 25357.749,E2 25357.749} C_VEL
LIN {X 0,Y 537.266,Z 348.586,A -85,B 0,C 180,E1 25357.139,E2 25357.139} C_VEL
LIN {X 0,Y 540.208,Z 351.098,A -85,B 0,C 180,E1 25356.318,E2 25356.318} C_VEL
LIN {X 0,Y 541.114,Z 351.924,A -85,B 0,C 180,E1 25356.071,E2 25356.071} C_VEL
LIN {X 0,Y 543.747,Z 355.699,A -85,B 0,C 180,E1 25355.328,E2 25355.328} C_VEL
LIN {X 0,Y 546.51,Z 358.169,A -85,B 0,C 180,E1 25354.622,E2 25354.622} C_VEL
LIN {X 0,Y 549.608,Z 362.3,A -85,B 0,C 180,E1 25353.821,E2 25353.821} C_VEL
LIN {X 0,Y 551.799,Z 364.442,A -85,B 0,C 180,E1 25353.295,E2 25353.295} C_VEL
LIN {X 0,Y 555.38,Z 368.907,A -85,B 0,C 180,E1 25352.439,E2 25352.439} C_VEL
LIN {X 0,Y 557.137,Z 370.799,A -85,B 0,C 180,E1 25352.039,E2 25352.039} C_VEL
LIN {X 0,Y 561.007,Z 375.35,A -85,B 0,C 180,E1 25351.176,E2 25351.176} C_VEL
LIN {X 0,Y 567.348,Z 383.446,A -85,B 0,C 180,E1 25349.82,E2 25349.82} C_VEL
LIN {X 0,Y 574.457,Z 392.134,A -85,B 0,C 180,E1 25348.405,E2 25348.405} C_VEL
LIN {X 0,Y 587.476,Z 409.322,A -85,B 0,C 180,E1 25346.005,E2 25346.005} C_VEL
LIN {X 0,Y 599.413,Z 425.985,A -85,B 0,C 180,E1 25343.997,E2 25343.997} C_VEL
LIN {X 0,Y 591.415,Z 637.487,A -85,B 0,C 180,E1 25340.883,E2 25340.883} C_VEL
LIN {X 0,Y 585.489,Z 799.296,A -85,B 0,C 180,E1 25338.522,E2 25338.522} C_VEL
LIN {X 0,Y 583.827,Z 823.702,A -85,B 0,C 180,E1 25338.065,E2 25338.065} C_VEL
LIN {X 0,Y 582.086,Z 842.944,A -85,B 0,C 180,E1 25337.598,E2 25337.598} C_VEL
LIN {X 0,Y 580.684,Z 850.472,A -85,B 0,C 180,E1 25337.467,E2 25337.467} C_VEL
LIN {X 0,Y 574.344,Z 869.614,A -85,B 0,C 180,E1 25337.311,E2 25337.311} C_VEL
LIN {X 0,Y 572.725,Z 876.83,A -85,B 0,C 180,E1 25337.125,E2 25337.125} C_VEL
LIN {X 0,Y 569.678,Z 898.478,A -85,B 0,C 180,E1 25336.269,E2 25336.269} C_VEL
LIN {X 0,Y 565.458,Z 924.925,A -85,B 0,C 180,E1 25335.015,E2 25335.015} C_VEL
LIN {X 0,Y 561.653,Z 946.073,A -85,B 0,C 180,E1 25333.828,E2 25333.828} C_VEL
LIN {X 0,Y 558.195,Z 964.011,A -85,B 0,C 180,E1 25332.686,E2 25332.686} C_VEL
LIN {X 0,Y 554.531,Z 981.984,A -85,B 0,C 180,E1 25331.401,E2 25331.401} C_VEL
LIN {X 0,Y 550.787,Z 999.605,A -85,B 0,C 180,E1 25329.988,E2 25329.988} C_VEL
LIN {X 0,Y 546.488,Z 1019.414,A -85,B 0,C 180,E1 25328.2,E2 25328.2} C_VEL
LIN {X 0,Y 541.729,Z 1040.541,A -85,B 0,C 180,E1 25326.004,E2 25326.004} C_VEL
LIN {X 0,Y 538.074,Z 1056.754,A -85,B 0,C 180,E1 25324.093,E2 25324.093} C_VEL
LIN {X 0,Y 534.865,Z 1071.216,A -85,B 0,C 180,E1 25322.193,E2 25322.193} C_VEL
LIN {X 0,Y 531.145,Z 1089.208,A -85,B 0,C 180,E1 25319.551,E2 25319.551} C_VEL
LIN {X 0,Y 528.159,Z 1104.216,A -85,B 0,C 180,E1 25317.023,E2 25317.023} C_VEL
LIN {X 0,Y 525.993,Z 1116.348,A -85,B 0,C 180,E1 25314.721,E2 25314.721} C_VEL
LIN {X 0,Y 524.156,Z 1127.671,A -85,B 0,C 180,E1 25312.301,E2 25312.301} C_VEL
LIN {X 0,Y 522.412,Z 1140.113,A -85,B 0,C 180,E1 25309.22,E2 25309.22} C_VEL
LIN {X 0,Y 521.38,Z 1149.011,A -85,B 0,C 180,E1 25306.603,E2 25306.603} C_VEL
LIN {X 0,Y 520.734,Z 1155.94,A -85,B 0,C 180,E1 25304.227,E2 25304.227} C_VEL
LIN {X 0,Y 520.312,Z 1161.986,A -85,B 0,C 180,E1 25301.753,E2 25301.753} C_VEL
LIN {X 0,Y 520.051,Z 1167.658,A -85,B 0,C 180,E1 25298.848,E2 25298.848} C_VEL
LIN {X 0,Y 519.944,Z 1171.587,A -85,B 0,C 180,E1 25295.96,E2 25295.96} C_VEL
LIN {X 0,Y 519.915,Z 1173.803,A -85,B 0,C 180,E1 25293.418,E2 25293.418} C_VEL
LIN {X 0,Y 519.91,Z 1174.771,A -85,B 0,C 180,E1 25291.102,E2 25291.102} C_VEL
LIN {X 0,Y 519.908,Z 1174.79,A -85,B 0,C 180,E1 25288.898,E2 25288.898} C_VEL
LIN {X 0,Y 519.912,Z 1173.859,A -85,B 0,C 180,E1 25286.582,E2 25286.582} C_VEL
LIN {X 0,Y 519.939,Z 1171.794,A -85,B 0,C 180,E1 25284.15,E2 25284.15} C_VEL
LIN {X 0,Y 520.037,Z 1168.147,A -85,B 0,C 180,E1 25281.375,E2 25281.375} C_VEL
LIN {X 0,Y 520.285,Z 1162.444,A -85,B 0,C 180,E1 25278.359,E2 25278.359} C_VEL
LIN {X 0,Y 520.716,Z 1156.181,A -85,B 0,C 180,E1 25275.772,E2 25275.772} C_VEL
LIN {X 0,Y 521.348,Z 1149.291,A -85,B 0,C 180,E1 25273.396,E2 25273.396} C_VEL
LIN {X 0,Y 522.265,Z 1141.236,A -85,B 0,C 180,E1 25271.007,E2 25271.007} C_VEL
LIN {X 0,Y 523.869,Z 1129.717,A -85,B 0,C 180,E1 25268.066,E2 25268.066} C_VEL
LIN {X 0,Y 525.852,Z 1117.167,A -85,B 0,C 180,E1 25265.355,E2 25265.355} C_VEL
LIN {X 0,Y 527.941,Z 1105.317,A -85,B 0,C 180,E1 25263.087,E2 25263.087} C_VEL
LIN {X 0,Y 530.427,Z 1092.521,A -85,B 0,C 180,E1 25260.9,E2 25260.9} C_VEL
LIN {X 0,Y 534.209,Z 1074.303,A -85,B 0,C 180,E1 25258.143,E2 25258.143} C_VEL
LIN {X 0,Y 537.796,Z 1057.987,A -85,B 0,C 180,E1 25255.971,E2 25255.971} C_VEL
LIN {X 0,Y 541.335,Z 1042.228,A -85,B 0,C 180,E1 25254.096,E2 25254.096} C_VEL
LIN {X 0,Y 545.547,Z 1023.632,A -85,B 0,C 180,E1 25252.123,E2 25252.123} C_VEL
LIN {X 0,Y 550.338,Z 1001.81,A -85,B 0,C 180,E1 25250.109,E2 25250.109} C_VEL
LIN {X 0,Y 554.181,Z 983.715,A -85,B 0,C 180,E1 25248.641,E2 25248.641} C_VEL
LIN {X 0,Y 557.83,Z 965.859,A -85,B 0,C 180,E1 25247.349,E2 25247.349} C_VEL
LIN {X 0,Y 561.38,Z 947.486,A -85,B 0,C 180,E1 25246.167,E2 25246.167} C_VEL
LIN {X 0,Y 565.039,Z 927.175,A -85,B 0,C 180,E1 25245.015,E2 25245.015} C_VEL
LIN {X 0,Y 569.384,Z 900.593,A -85,B 0,C 180,E1 25243.73,E2 25243.73} C_VEL
LIN {X 0,Y 572.585,Z 877.992,A -85,B 0,C 180,E1 25242.827,E2 25242.827} C_VEL
LIN {X 0,Y 575.215,Z 856.653,A -85,B 0,C 180,E1 25242.111,E2 25242.111} C_VEL
LIN {X 0,Y 577.436,Z 835.503,A -85,B 0,C 180,E1 25241.526,E2 25241.526} C_VEL
LIN {X 0,Y 579.391,Z 812.58,A -85,B 0,C 180,E1 25241.022,E2 25241.022} C_VEL
LIN {X 0,Y 581.256,Z 776.826,A -85,B 0,C 180,E1 25240.448,E2 25240.448} C_VEL
LIN {X 0,Y 589.676,Z 553.529,A -85,B 0,C 180,E1 25237.18,E2 25237.18} C_VEL
LIN {X 0,Y 594.583,Z 430.338,A -85,B 0,C 180,E1 25235.345,E2 25235.345} C_VEL
LIN {X 0,Y 582.556,Z 413.498,A -85,B 0,C 180,E1 25233.256,E2 25233.256} C_VEL
LIN {X 0,Y 573.415,Z 401.46,A -85,B 0,C 180,E1 25231.542,E2 25231.542} C_VEL
LIN {X 0,Y 566.344,Z 392.422,A -85,B 0,C 180,E1 25230.123,E2 25230.123} C_VEL
LIN {X 0,Y 561.471,Z 386.348,A -85,B 0,C 180,E1 25229.089,E2 25229.089} C_VEL
LIN {X 0,Y 557.583,Z 381.533,A -85,B 0,C 180,E1 25228.228,E2 25228.228} C_VEL
LIN {X 0,Y 553.452,Z 376.491,A -85,B 0,C 180,E1 25227.273,E2 25227.273} C_VEL
LIN {X 0,Y 549.641,Z 371.909,A -85,B 0,C 180,E1 25226.352,E2 25226.352} C_VEL
LIN {X 0,Y 544.86,Z 366.408,A -85,B 0,C 180,E1 25225.14,E2 25225.14} C_VEL
LIN {X 0,Y 543.584,Z 364.71,A -85,B 0,C 180,E1 25224.796,E2 25224.796} C_VEL
LIN {X 0,Y 540.102,Z 361.135,A -85,B 0,C 180,E1 25223.861,E2 25223.861} C_VEL
LIN {X 0,Y 538.574,Z 358.806,A -85,B 0,C 180,E1 25223.41,E2 25223.41} C_VEL
LIN {X 0,Y 535.15,Z 355.796,A -85,B 0,C 180,E1 25222.435,E2 25222.435} C_VEL
LIN {X 0,Y 533.193,Z 352.498,A -85,B 0,C 180,E1 25221.796,E2 25221.796} C_VEL
LIN {X 0,Y 529.874,Z 350.08,A -85,B 0,C 180,E1 25220.779,E2 25220.779} C_VEL
LIN {X 0,Y 527.899,Z 346.962,A -85,B 0,C 180,E1 25220.078,E2 25220.078} C_VEL
LIN {X 0,Y 527.43,Z 345.902,A -85,B 0,C 180,E1 25219.895,E2 25219.895} C_VEL
LIN {X 0,Y 524.053,Z 343.953,A -85,B 0,C 180,E1 25218.754,E2 25218.754} C_VEL
LIN {X 0,Y 522.185,Z 341.249,A -85,B 0,C 180,E1 25218.014,E2 25218.014} C_VEL
LIN {X 0,Y 521.675,Z 339.25,A -85,B 0,C 180,E1 25217.719,E2 25217.719} C_VEL
LIN {X 0,Y 521.663,Z 339.186,A -85,B 0,C 180,E1 25214.202,E2 25214.202} C_VEL
LIN {X 0,Y 521.731,Z 339.216,A -85,B 0,C 180,E1 25210.937,E2 25210.937} C_VEL
LIN {X 0,Y 521.673,Z 339.195,A -85,B 0,C 180,E1 25207.6,E2 25207.6} C_VEL
LIN {X 0,Y 521.686,Z 339.198,A -85,B 0,C 180,E1 25204.177,E2 25204.177} C_VEL
LIN {X 0,Y 521.742,Z 339.209,A -85,B 0,C 180,E1 25200.769,E2 25200.769} C_VEL
LIN {X 0,Y 521.68,Z 339.186,A -85,B 0,C 180,E1 25197.473,E2 25197.473} C_VEL
LIN {X 0,Y 521.711,Z 339.237,A -85,B 0,C 180,E1 25194.06,E2 25194.06} C_VEL
LIN {X 0,Y 521.714,Z 339.176,A -85,B 0,C 180,E1 25190.847,E2 25190.847} C_VEL
LIN {X 0,Y 521.695,Z 339.239,A -85,B 0,C 180,E1 25187.492,E2 25187.492} C_VEL
LIN {X 0,Y 521.742,Z 339.184,A -85,B 0,C 180,E1 25184.159,E2 25184.159} C_VEL
LIN {X 0,Y 521.733,Z 339.394,A -85,B 0,C 180,E1 25182.892,E2 25182.892} C_VEL
LIN {X 0,Y 522.413,Z 341.575,A -85,B 0,C 180,E1 25182.311,E2 25182.311} C_VEL
LIN {X 0,Y 524.375,Z 344.25,A -85,B 0,C 180,E1 25181.547,E2 25181.547} C_VEL
LIN {X 0,Y 526.705,Z 345.982,A -85,B 0,C 180,E1 25180.741,E2 25180.741} C_VEL
LIN {X 0,Y 531.026,Z 351.187,A -85,B 0,C 180,E1 25179.268,E2 25179.268} C_VEL
LIN {X 0,Y 532.597,Z 353.255,A -85,B 0,C 180,E1 25178.756,E2 25178.756} C_VEL
LIN {X 0,Y 536.842,Z 358.093,A -85,B 0,C 180,E1 25177.467,E2 25177.467} C_VEL
LIN {X 0,Y 540.566,Z 362.734,A -85,B 0,C 180,E1 25176.393,E2 25176.393} C_VEL
LIN {X 0,Y 546.872,Z 370.722,A -85,B 0,C 180,E1 25174.698,E2 25174.698} C_VEL
LIN {X 0,Y 551.007,Z 375.99,A -85,B 0,C 180,E1 25173.661,E2 25173.661} C_VEL
LIN {X 0,Y 555.286,Z 381.567,A -85,B 0,C 180,E1 25172.637,E2 25172.637} C_VEL
LIN {X 0,Y 560.45,Z 388.341,A -85,B 0,C 180,E1 25171.465,E2 25171.465} C_VEL
LIN {X 0,Y 569.55,Z 400.719,A -85,B 0,C 180,E1 25169.537,E2 25169.537} C_VEL
LIN {X 0,Y 581.812,Z 418.354,A -85,B 0,C 180,E1 25167.165,E2 25167.165} C_VEL
LIN {X 0,Y 594.182,Z 437.407,A -85,B 0,C 180,E1 25164.982,E2 25164.982} C_VEL
LIN {X 0,Y 594.757,Z 438.72,A -85,B 0,C 180,E1 25164.876,E2 25164.876} C_VEL
LIN {X 0,Y 586.309,Z 655.157,A -85,B 0,C 180,E1 25161.675,E2 25161.675} C_VEL
LIN {X 0,Y 579.948,Z 824.343,A -85,B 0,C 180,E1 25159.195,E2 25159.195} C_VEL
LIN {X 0,Y 578.127,Z 849.507,A -85,B 0,C 180,E1 25158.731,E2 25158.731} C_VEL
LIN {X 0,Y 575.296,Z 877.611,A -85,B 0,C 180,E1 25158.021,E2 25158.021} C_VEL
LIN {X 0,Y 572.605,Z 899.653,A -85,B 0,C 180,E1 25157.318,E2 25157.318} C_VEL
LIN {X 0,Y 569.754,Z 920.284,A -85,B 0,C 180,E1 25156.532,E2 25156.532} C_VEL
LIN {X 0,Y 566.584,Z 940.86,A -85,B 0,C 180,E1 25155.619,E2 25155.619} C_VEL
LIN {X 0,Y 562.385,Z 965.923,A -85,B 0,C 180,E1 25154.323,E2 25154.323} C_VEL
LIN {X 0,Y 557.928,Z 989.671,A -85,B 0,C 180,E1 25152.862,E2 25152.862} C_VEL
LIN {X 0,Y 554.107,Z 1009.016,A -85,B 0,C 180,E1 25151.507,E2 25151.507} C_VEL
LIN {X 0,Y 550.281,Z 1027.729,A -85,B 0,C 180,E1 25150.032,E2 25150.032} C_VEL
LIN {X 0,Y 545.831,Z 1049.226,A -85,B 0,C 180,E1 25148.121,E2 25148.121} C_VEL
LIN {X 0,Y 541.305,Z 1070.151,A -85,B 0,C 180,E1 25145.972,E2 25145.972} C_VEL
LIN {X 0,Y 537.942,Z 1085.987,A -85,B 0,C 180,E1 25144.147,E2 25144.147} C_VEL
LIN {X 0,Y 534.752,Z 1101.219,A -85,B 0,C 180,E1 25142.2,E2 25142.2} C_VEL
LIN {X 0,Y 531.944,Z 1114.909,A -85,B 0,C 180,E1 25140.248,E2 25140.248} C_VEL
LIN {X 0,Y 528.759,Z 1131.273,A -85,B 0,C 180,E1 25137.599,E2 25137.599} C_VEL
LIN {X 0,Y 526.245,Z 1144.837,A -85,B 0,C 180,E1 25135.068,E2 25135.068} C_VEL
LIN {X 0,Y 524.441,Z 1155.769,A -85,B 0,C 180,E1 25132.769,E2 25132.769} C_VEL
LIN {X 0,Y 522.963,Z 1165.894,A -85,B 0,C 180,E1 25130.363,E2 25130.363} C_VEL
LIN {X 0,Y 521.631,Z 1176.674,A -85,B 0,C 180,E1 25127.399,E2 25127.399} C_VEL
LIN {X 0,Y 520.805,Z 1185.152,A -85,B 0,C 180,E1 25124.566,E2 25124.566} C_VEL
LIN {X 0,Y 520.345,Z 1191.325,A -85,B 0,C 180,E1 25122.09,E2 25122.09} C_VEL
LIN {X 0,Y 520.088,Z 1196.542,A -85,B 0,C 180,E1 25119.506,E2 25119.506} C_VEL
LIN {X 0,Y 519.955,Z 1201.053,A -85,B 0,C 180,E1 25116.515,E2 25116.515} C_VEL
LIN {X 0,Y 519.913,Z 1203.627,A -85,B 0,C 180,E1 25113.749,E2 25113.749} C_VEL
LIN {X 0,Y 519.914,Z 1204.735,A -85,B 0,C 180,E1 25111.322,E2 25111.322} C_VEL
LIN {X 0,Y 519.909,Z 1204.803,A -85,B 0,C 180,E1 25109.008,E2 25109.008} C_VEL
LIN {X 0,Y 519.916,Z 1203.898,A -85,B 0,C 180,E1 25106.693,E2 25106.693} C_VEL
LIN {X 0,Y 519.937,Z 1201.861,A -85,B 0,C 180,E1 25104.261,E2 25104.261} C_VEL
LIN {X 0,Y 520.022,Z 1198.401,A -85,B 0,C 180,E1 25101.597,E2 25101.597} C_VEL
LIN {X 0,Y 520.256,Z 1192.832,A -85,B 0,C 180,E1 25098.575,E2 25098.575} C_VEL
LIN {X 0,Y 520.713,Z 1186.309,A -85,B 0,C 180,E1 25095.865,E2 25095.865} C_VEL
LIN {X 0,Y 521.322,Z 1179.503,A -85,B 0,C 180,E1 25093.51,E2 25093.51} C_VEL
LIN {X 0,Y 522.275,Z 1171.205,A -85,B 0,C 180,E1 25091.043,E2 25091.043} C_VEL
LIN {X 0,Y 523.851,Z 1159.893,A -85,B 0,C 180,E1 25088.149,E2 25088.149} C_VEL
LIN {X 0,Y 525.859,Z 1147.136,A -85,B 0,C 180,E1 25085.392,E2 25085.392} C_VEL
LIN {X 0,Y 527.943,Z 1135.319,A -85,B 0,C 180,E1 25083.132,E2 25083.132} C_VEL
LIN {X 0,Y 530.483,Z 1122.266,A -85,B 0,C 180,E1 25080.904,E2 25080.904} C_VEL
LIN {X 0,Y 533.916,Z 1105.513,A -85,B 0,C 180,E1 25078.375,E2 25078.375} C_VEL
LIN {X 0,Y 537.535,Z 1087.867,A -85,B 0,C 180,E1 25076.081,E2 25076.081} C_VEL
LIN {X 0,Y 540.861,Z 1072.171,A -85,B 0,C 180,E1 25074.251,E2 25074.251} C_VEL
LIN {X 0,Y 544.407,Z 1055.571,A -85,B 0,C 180,E1 25072.508,E2 25072.508} C_VEL
LIN {X 0,Y 548.956,Z 1034.439,A -85,B 0,C 180,E1 25070.531,E2 25070.531} C_VEL
LIN {X 0,Y 553.523,Z 1012.004,A -85,B 0,C 180,E1 25068.718,E2 25068.718} C_VEL
LIN {X 0,Y 557.298,Z 992.961,A -85,B 0,C 180,E1 25067.359,E2 25067.359} C_VEL
LIN {X 0,Y 560.689,Z 975.024,A -85,B 0,C 180,E1 25066.219,E2 25066.219} C_VEL
LIN {X 0,Y 564.093,Z 955.811,A -85,B 0,C 180,E1 25065.134,E2 25065.134} C_VEL
LIN {X 0,Y 567.683,Z 934.028,A -85,B 0,C 180,E1 25064.06,E2 25064.06} C_VEL
LIN {X 0,Y 571.744,Z 906.332,A -85,B 0,C 180,E1 25062.92,E2 25062.92} C_VEL
LIN {X 0,Y 574.609,Z 883.528,A -85,B 0,C 180,E1 25062.156,E2 25062.156} C_VEL
LIN {X 0,Y 576.911,Z 862.051,A -85,B 0,C 180,E1 25061.564,E2 25061.564} C_VEL
LIN {X 0,Y 578.836,Z 840.5,A -85,B 0,C 180,E1 25061.091,E2 25061.091} C_VEL
LIN {X 0,Y 580.456,Z 814.594,A -85,B 0,C 180,E1 25060.651,E2 25060.651} C_VEL
LIN {X 0,Y 588.732,Z 590.899,A -85,B 0,C 180,E1 25057.382,E2 25057.382} C_VEL
LIN {X 0,Y 594.652,Z 438.201,A -85,B 0,C 180,E1 25055.104,E2 25055.104} C_VEL
LIN {X 0,Y 583.066,Z 420.379,A -85,B 0,C 180,E1 25053.077,E2 25053.077} C_VEL
LIN {X 0,Y 572.17,Z 404.437,A -85,B 0,C 180,E1 25051.003,E2 25051.003} C_VEL
LIN {X 0,Y 561.445,Z 389.628,A -85,B 0,C 180,E1 25048.77,E2 25048.77} C_VEL
LIN {X 0,Y 556.43,Z 383.126,A -85,B 0,C 180,E1 25047.65,E2 25047.65} C_VEL
LIN {X 0,Y 552.402,Z 377.838,A -85,B 0,C 180,E1 25046.702,E2 25046.702} C_VEL
LIN {X 0,Y 548.02,Z 372.189,A -85,B 0,C 180,E1 25045.621,E2 25045.621} C_VEL
LIN {X 0,Y 544.258,Z 367.47,A -85,B 0,C 180,E1 25044.648,E2 25044.648} C_VEL
LIN {X 0,Y 540.464,Z 362.648,A -85,B 0,C 180,E1 25043.612,E2 25043.612} C_VEL
LIN {X 0,Y 536.821,Z 358.072,A -85,B 0,C 180,E1 25042.563,E2 25042.563} C_VEL
LIN {X 0,Y 532.096,Z 352.507,A -85,B 0,C 180,E1 25041.12,E2 25041.12} C_VEL
LIN {X 0,Y 530.904,Z 351.088,A -85,B 0,C 180,E1 25040.737,E2 25040.737} C_VEL
LIN {X 0,Y 526.653,Z 345.904,A -85,B 0,C 180,E1 25039.29,E2 25039.29} C_VEL
LIN {X 0,Y 523.255,Z 343.017,A -85,B 0,C 180,E1 25038.091,E2 25038.091} C_VEL
LIN {X 0,Y 521.965,Z 340.365,A -85,B 0,C 180,E1 25037.456,E2 25037.456} C_VEL
LIN {X 0,Y 521.712,Z 339.228,A -85,B 0,C 180,E1 25037.052,E2 25037.052} C_VEL
LIN {X 0,Y 521.747,Z 339.188,A -85,B 0,C 180,E1 25033.689,E2 25033.689} C_VEL
LIN {X 0,Y 521.693,Z 339.196,A -85,B 0,C 180,E1 25030.379,E2 25030.379} C_VEL
LIN {X 0,Y 521.707,Z 339.225,A -85,B 0,C 180,E1 25026.903,E2 25026.903} C_VEL
LIN {X 0,Y 521.725,Z 339.177,A -85,B 0,C 180,E1 25023.626,E2 25023.626} C_VEL
LIN {X 0,Y 521.687,Z 339.247,A -85,B 0,C 180,E1 25020.329,E2 25020.329} C_VEL
LIN {X 0,Y 521.723,Z 339.174,A -85,B 0,C 180,E1 25017.034,E2 25017.034} C_VEL
LIN {X 0,Y 521.697,Z 339.247,A -85,B 0,C 180,E1 25013.728,E2 25013.728} C_VEL
LIN {X 0,Y 521.674,Z 339.185,A -85,B 0,C 180,E1 25010.289,E2 25010.289} C_VEL
LIN {X 0,Y 521.735,Z 339.21,A -85,B 0,C 180,E1 25006.93,E2 25006.93} C_VEL
LIN {X 0,Y 521.669,Z 339.2,A -85,B 0,C 180,E1 25003.749,E2 25003.749} C_VEL
LIN {X 0,Y 521.698,Z 339.433,A -85,B 0,C 180,E1 25002.084,E2 25002.084} C_VEL
LIN {X 0,Y 522.612,Z 342.118,A -85,B 0,C 180,E1 25001.655,E2 25001.655} C_VEL
LIN {X 0,Y 525.012,Z 344.718,A -85,B 0,C 180,E1 25000.763,E2 25000.763} C_VEL
LIN {X 0,Y 527.591,Z 346.123,A -85,B 0,C 180,E1 24999.909,E2 24999.909} C_VEL
LIN {X 0,Y 529.361,Z 349.461,A -85,B 0,C 180,E1 24999.258,E2 24999.258} C_VEL
LIN {X 0,Y 532.454,Z 352.143,A -85,B 0,C 180,E1 24998.288,E2 24998.288} C_VEL
LIN {X 0,Y 533.389,Z 352.821,A -85,B 0,C 180,E1 24998.009,E2 24998.009} C_VEL
LIN {X 0,Y 535.706,Z 356.444,A -85,B 0,C 180,E1 24997.271,E2 24997.271} C_VEL
LIN {X 0,Y 539.07,Z 359.45,A -85,B 0,C 180,E1 24996.323,E2 24996.323} C_VEL
LIN {X 0,Y 542.06,Z 363.429,A -85,B 0,C 180,E1 24995.478,E2 24995.478} C_VEL
LIN {X 0,Y 544.408,Z 365.676,A -85,B 0,C 180,E1 24994.867,E2 24994.867} C_VEL
LIN {X 0,Y 547.883,Z 370.036,A -85,B 0,C 180,E1 24993.965,E2 24993.965} C_VEL
LIN {X 0,Y 549.646,Z 371.933,A -85,B 0,C 180,E1 24993.532,E2 24993.532} C_VEL
LIN {X 0,Y 553.414,Z 376.46,A -85,B 0,C 180,E1 24992.624,E2 24992.624} C_VEL
LIN {X 0,Y 559.915,Z 384.393,A -85,B 0,C 180,E1 24991.144,E2 24991.144} C_VEL
LIN {X 0,Y 564.739,Z 390.469,A -85,B 0,C 180,E1 24990.105,E2 24990.105} C_VEL
LIN {X 0,Y 571.886,Z 399.366,A -85,B 0,C 180,E1 24988.657,E2 24988.657} C_VEL
LIN {X 0,Y 584.077,Z 415.552,A -85,B 0,C 180,E1 24986.371,E2 24986.371} C_VEL
LIN {X 0,Y 594.58,Z 430.383,A -85,B 0,C 180,E1 24984.559,E2 24984.559} C_VEL
LIN {X 0,Y 586.146,Z 644.375,A -85,B 0,C 180,E1 24981.393,E2 24981.393} C_VEL
LIN {X 0,Y 580.216,Z 799.62,A -85,B 0,C 180,E1 24979.114,E2 24979.114} C_VEL
LIN {X 0,Y 578.488,Z 824.149,A -85,B 0,C 180,E1 24978.653,E2 24978.653} C_VEL
LIN {X 0,Y 575.747,Z 852.072,A -85,B 0,C 180,E1 24977.937,E2 24977.937} C_VEL
LIN {X 0,Y 573.094,Z 873.965,A -85,B 0,C 180,E1 24977.228,E2 24977.228} C_VEL
LIN {X 0,Y 572.725,Z 876.83,A -85,B 0,C 180,E1 24977.125,E2 24977.125} C_VEL
LIN {X 0,Y 571.087,Z 884.363,A -85,B 0,C 180,E1 24976.926,E2 24976.926} C_VEL
LIN {X 0,Y 563.883,Z 903.89,A -85,B 0,C 180,E1 24976.586,E2 24976.586} C_VEL
LIN {X 0,Y 562.314,Z 909.896,A -85,B 0,C 180,E1 24976.361,E2 24976.361} C_VEL
LIN {X 0,Y 558.775,Z 930.284,A -85,B 0,C 180,E1 24975.331,E2 24975.331} C_VEL
LIN {X 0,Y 555.086,Z 949.917,A -85,B 0,C 180,E1 24974.194,E2 24974.194} C_VEL
LIN {X 0,Y 551.047,Z 969.91,A -85,B 0,C 180,E1 24972.877,E2 24972.877} C_VEL
LIN {X 0,Y 545.832,Z 993.947,A -85,B 0,C 180,E1 24971.049,E2 24971.049} C_VEL
LIN {X 0,Y 541.465,Z 1013.089,A -85,B 0,C 180,E1 24969.368,E2 24969.368} C_VEL
LIN {X 0,Y 537.595,Z 1029.737,A -85,B 0,C 180,E1 24967.727,E2 24967.727} C_VEL
LIN {X 0,Y 533.714,Z 1046.314,A -85,B 0,C 180,E1 24965.9,E2 24965.9} C_VEL
LIN {X 0,Y 529.221,Z 1065.677,A -85,B 0,C 180,E1 24963.482,E2 24963.482} C_VEL
LIN {X 0,Y 525.676,Z 1081.056,A -85,B 0,C 180,E1 24961.282,E2 24961.282} C_VEL
LIN {X 0,Y 522.764,Z 1094.153,A -85,B 0,C 180,E1 24959.191,E2 24959.191} C_VEL
LIN {X 0,Y 520.078,Z 1107.392,A -85,B 0,C 180,E1 24956.859,E2 24956.859} C_VEL
LIN {X 0,Y 517.524,Z 1121.461,A -85,B 0,C 180,E1 24954.057,E2 24954.057} C_VEL
LIN {X 0,Y 515.546,Z 1133.43,A -85,B 0,C 180,E1 24951.264,E2 24951.264} C_VEL
LIN {X 0,Y 514.313,Z 1142.138,A -85,B 0,C 180,E1 24948.945,E2 24948.945} C_VEL
LIN {X 0,Y 513.372,Z 1150.072,A -85,B 0,C 180,E1 24946.52,E2 24946.52} C_VEL
LIN {X 0,Y 512.677,Z 1157.454,A -85,B 0,C 180,E1 24943.88,E2 24943.88} C_VEL
LIN {X 0,Y 512.197,Z 1164.578,A -85,B 0,C 180,E1 24940.687,E2 24940.687} C_VEL
LIN {X 0,Y 512.014,Z 1168.996,A -85,B 0,C 180,E1 24938.067,E2 24938.067} C_VEL
LIN {X 0,Y 511.936,Z 1172.04,A -85,B 0,C 180,E1 24935.604,E2 24935.604} C_VEL
LIN {X 0,Y 511.913,Z 1174.004,A -85,B 0,C 180,E1 24933.135,E2 24933.135} C_VEL
LIN {X 0,Y 511.897,Z 1174.862,A -85,B 0,C 180,E1 24930.671,E2 24930.671} C_VEL
LIN {X 0,Y 511.912,Z 1174.586,A -85,B 0,C 180,E1 24927.873,E2 24927.873} C_VEL
LIN {X 0,Y 511.925,Z 1172.586,A -85,B 0,C 180,E1 24924.845,E2 24924.845} C_VEL
LIN {X 0,Y 511.99,Z 1169.581,A -85,B 0,C 180,E1 24922.256,E2 24922.256} C_VEL
LIN {X 0,Y 512.145,Z 1165.568,A -85,B 0,C 180,E1 24919.767,E2 24919.767} C_VEL
LIN {X 0,Y 512.469,Z 1160.15,A -85,B 0,C 180,E1 24917.149,E2 24917.149} C_VEL
LIN {X 0,Y 513.16,Z 1152.114,A -85,B 0,C 180,E1 24914.054,E2 24914.054} C_VEL
LIN {X 0,Y 514.178,Z 1143.206,A -85,B 0,C 180,E1 24911.27,E2 24911.27} C_VEL
LIN {X 0,Y 515.425,Z 1134.231,A -85,B 0,C 180,E1 24908.85,E2 24908.85} C_VEL
LIN {X 0,Y 517.076,Z 1123.9,A -85,B 0,C 180,E1 24906.405,E2 24906.405} C_VEL
LIN {X 0,Y 519.678,Z 1109.651,A -85,B 0,C 180,E1 24903.469,E2 24903.469} C_VEL
LIN {X 0,Y 522.499,Z 1095.333,A -85,B 0,C 180,E1 24900.918,E2 24900.918} C_VEL
LIN {X 0,Y 525.376,Z 1082.349,A -85,B 0,C 180,E1 24898.825,E2 24898.825} C_VEL
LIN {X 0,Y 528.742,Z 1067.675,A -85,B 0,C 180,E1 24896.705,E2 24896.705} C_VEL
LIN {X 0,Y 533.447,Z 1047.492,A -85,B 0,C 180,E1 24894.146,E2 24894.146} C_VEL
LIN {X 0,Y 537.443,Z 1030.39,A -85,B 0,C 180,E1 24892.251,E2 24892.251} C_VEL
LIN {X 0,Y 541.28,Z 1013.886,A -85,B 0,C 180,E1 24890.616,E2 24890.616} C_VEL
LIN {X 0,Y 545.477,Z 995.473,A -85,B 0,C 180,E1 24888.989,E2 24888.989} C_VEL
LIN {X 0,Y 550.664,Z 971.825,A -85,B 0,C 180,E1 24887.164,E2 24887.164} C_VEL
LIN {X 0,Y 554.867,Z 951.039,A -85,B 0,C 180,E1 24885.784,E2 24885.784} C_VEL
LIN {X 0,Y 558.568,Z 931.421,A -85,B 0,C 180,E1 24884.64,E2 24884.64} C_VEL
LIN {X 0,Y 562.085,Z 911.292,A -85,B 0,C 180,E1 24883.616,E2 24883.616} C_VEL
LIN {X 0,Y 565.555,Z 889.362,A -85,B 0,C 180,E1 24882.654,E2 24882.654} C_VEL
LIN {X 0,Y 569.333,Z 861.347,A -85,B 0,C 180,E1 24881.647,E2 24881.647} C_VEL
LIN {X 0,Y 571.845,Z 838.826,A -85,B 0,C 180,E1 24881.002,E2 24881.002} C_VEL
LIN {X 0,Y 573.77,Z 817.516,A -85,B 0,C 180,E1 24880.512,E2 24880.512} C_VEL
LIN {X 0,Y 575.276,Z 795.305,A -85,B 0,C 180,E1 24880.118,E2 24880.118} C_VEL
LIN {X 0,Y 584.055,Z 573.682,A -85,B 0,C 180,E1 24876.849,E2 24876.849} C_VEL
LIN {X 0,Y 589.748,Z 434.529,A -85,B 0,C 180,E1 24874.76,E2 24874.76} C_VEL
LIN {X 0,Y 578.721,Z 419.167,A -85,B 0,C 180,E1 24872.796,E2 24872.796} C_VEL
LIN {X 0,Y 570.059,Z 407.583,A -85,B 0,C 180,E1 24871.131,E2 24871.131} C_VEL
LIN {X 0,Y 563.407,Z 399.053,A -85,B 0,C 180,E1 24869.767,E2 24869.767} C_VEL
LIN {X 0,Y 555.591,Z 389.115,A -85,B 0,C 180,E1 24868.045,E2 24868.045} C_VEL
LIN {X 0,Y 551.029,Z 383.616,A -85,B 0,C 180,E1 24866.978,E2 24866.978} C_VEL
LIN {X 0,Y 547.039,Z 378.64,A -85,B 0,C 180,E1 24865.991,E2 24865.991} C_VEL
LIN {X 0,Y 542.775,Z 373.836,A -85,B 0,C 180,E1 24864.894,E2 24864.894} C_VEL
LIN {X 0,Y 541.326,Z 371.967,A -85,B 0,C 180,E1 24864.499,E2 24864.499} C_VEL
LIN {X 0,Y 537.733,Z 368.026,A -85,B 0,C 180,E1 24863.507,E2 24863.507} C_VEL
LIN {X 0,Y 536.375,Z 366.16,A -85,B 0,C 180,E1 24863.104,E2 24863.104} C_VEL
LIN {X 0,Y 532.781,Z 362.618,A -85,B 0,C 180,E1 24862.046,E2 24862.046} C_VEL
LIN {X 0,Y 531.234,Z 360.055,A -85,B 0,C 180,E1 24861.533,E2 24861.533} C_VEL
LIN {X 0,Y 527.826,Z 357.276,A -85,B 0,C 180,E1 24860.457,E2 24860.457} C_VEL
LIN {X 0,Y 525.54,Z 353.563,A -85,B 0,C 180,E1 24859.622,E2 24859.622} C_VEL
LIN {X 0,Y 521.965,Z 351.073,A -85,B 0,C 180,E1 24858.368,E2 24858.368} C_VEL
LIN {X 0,Y 520.113,Z 347.979,A -85,B 0,C 180,E1 24857.596,E2 24857.596} C_VEL
LIN {X 0,Y 519.708,Z 346.994,A -85,B 0,C 180,E1 24857.408,E2 24857.408} C_VEL
LIN {X 0,Y 516.117,Z 344.967,A -85,B 0,C 180,E1 24855.968,E2 24855.968} C_VEL
LIN {X 0,Y 514.327,Z 342.225,A -85,B 0,C 180,E1 24855.1,E2 24855.1} C_VEL
LIN {X 0,Y 513.76,Z 340.165,A -85,B 0,C 180,E1 24854.707,E2 24854.707} C_VEL
LIN {X 0,Y 513.75,Z 340.231,A -85,B 0,C 180,E1 24851.45,E2 24851.45} C_VEL
LIN {X 0,Y 513.731,Z 340.173,A -85,B 0,C 180,E1 24848.056,E2 24848.056} C_VEL
LIN {X 0,Y 513.796,Z 340.199,A -85,B 0,C 180,E1 24844.8,E2 24844.8} C_VEL
LIN {X 0,Y 513.741,Z 340.181,A -85,B 0,C 180,E1 24841.45,E2 24841.45} C_VEL
LIN {X 0,Y 513.751,Z 340.182,A -85,B 0,C 180,E1 24837.992,E2 24837.992} C_VEL
LIN {X 0,Y 513.806,Z 340.2,A -85,B 0,C 180,E1 24834.528,E2 24834.528} C_VEL
LIN {X 0,Y 513.75,Z 340.169,A -85,B 0,C 180,E1 24831.268,E2 24831.268} C_VEL
LIN {X 0,Y 513.763,Z 340.232,A -85,B 0,C 180,E1 24827.678,E2 24827.678} C_VEL
LIN {X 0,Y 513.783,Z 340.368,A -85,B 0,C 180,E1 24825.647,E2 24825.647} C_VEL
LIN {X 0,Y 514.655,Z 342.987,A -85,B 0,C 180,E1 24825.14,E2 24825.14} C_VEL
LIN {X 0,Y 517.286,Z 345.845,A -85,B 0,C 180,E1 24823.954,E2 24823.954} C_VEL
LIN {X 0,Y 519.709,Z 347.272,A -85,B 0,C 180,E1 24822.996,E2 24822.996} C_VEL
LIN {X 0,Y 522.276,Z 351.383,A -85,B 0,C 180,E1 24821.932,E2 24821.932} C_VEL
LIN {X 0,Y 525.064,Z 353.695,A -85,B 0,C 180,E1 24820.938,E2 24820.938} C_VEL
LIN {X 0,Y 529.431,Z 358.874,A -85,B 0,C 180,E1 24819.434,E2 24819.434} C_VEL
LIN {X 0,Y 533.761,Z 364.197,A -85,B 0,C 180,E1 24818.055,E2 24818.055} C_VEL
LIN {X 0,Y 538.893,Z 370.444,A -85,B 0,C 180,E1 24816.547,E2 24816.547} C_VEL
LIN {X 0,Y 548.282,Z 382.587,A -85,B 0,C 180,E1 24814.044,E2 24814.044} C_VEL
LIN {X 0,Y 556.663,Z 393.618,A -85,B 0,C 180,E1 24812.043,E2 24812.043} C_VEL
LIN {X 0,Y 566.666,Z 407.431,A -85,B 0,C 180,E1 24809.867,E2 24809.867} C_VEL
LIN {X 0,Y 577.866,Z 423.77,A -85,B 0,C 180,E1 24807.649,E2 24807.649} C_VEL
LIN {X 0,Y 587.377,Z 438.446,A -85,B 0,C 180,E1 24805.911,E2 24805.911} C_VEL
LIN {X 0,Y 589.975,Z 442.634,A -85,B 0,C 180,E1 24805.455,E2 24805.455} C_VEL
LIN {X 0,Y 581.199,Z 658.669,A -85,B 0,C 180,E1 24802.243,E2 24802.243} C_VEL
LIN {X 0,Y 574.721,Z 824.066,A -85,B 0,C 180,E1 24799.803,E2 24799.803} C_VEL
LIN {X 0,Y 572.826,Z 849.417,A -85,B 0,C 180,E1 24799.334,E2 24799.334} C_VEL
LIN {X 0,Y 569.887,Z 877.506,A -85,B 0,C 180,E1 24798.623,E2 24798.623} C_VEL
LIN {X 0,Y 567.121,Z 899.392,A -85,B 0,C 180,E1 24797.922,E2 24797.922} C_VEL
LIN {X 0,Y 564.222,Z 919.611,A -85,B 0,C 180,E1 24797.152,E2 24797.152} C_VEL
LIN {X 0,Y 560.939,Z 940.137,A -85,B 0,C 180,E1 24796.241,E2 24796.241} C_VEL
LIN {X 0,Y 556.651,Z 964.756,A -85,B 0,C 180,E1 24794.968,E2 24794.968} C_VEL
LIN {X 0,Y 551.996,Z 988.709,A -85,B 0,C 180,E1 24793.496,E2 24793.496} C_VEL
LIN {X 0,Y 547.947,Z 1008.395,A -85,B 0,C 180,E1 24792.112,E2 24792.112} C_VEL
LIN {X 0,Y 544.022,Z 1026.794,A -85,B 0,C 180,E1 24790.656,E2 24790.656} C_VEL
LIN {X 0,Y 539.725,Z 1046.485,A -85,B 0,C 180,E1 24788.903,E2 24788.903} C_VEL
LIN {X 0,Y 534.745,Z 1068.846,A -85,B 0,C 180,E1 24786.617,E2 24786.617} C_VEL
LIN {X 0,Y 531.104,Z 1085.147,A -85,B 0,C 180,E1 24784.727,E2 24784.727} C_VEL
LIN {X 0,Y 527.818,Z 1100.083,A -85,B 0,C 180,E1 24782.805,E2 24782.805} C_VEL
LIN {X 0,Y 524.674,Z 1114.725,A -85,B 0,C 180,E1 24780.712,E2 24780.712} C_VEL
LIN {X 0,Y 521.433,Z 1130.844,A -85,B 0,C 180,E1 24778.104,E2 24778.104} C_VEL
LIN {X 0,Y 518.67,Z 1144.835,A -85,B 0,C 180,E1 24775.46,E2 24775.46} C_VEL
LIN {X 0,Y 516.758,Z 1155.767,A -85,B 0,C 180,E1 24773.127,E2 24773.127} C_VEL
LIN {X 0,Y 515.187,Z 1165.893,A -85,B 0,C 180,E1 24770.684,E2 24770.684} C_VEL
LIN {X 0,Y 513.763,Z 1176.675,A -85,B 0,C 180,E1 24767.674,E2 24767.674} C_VEL
LIN {X 0,Y 512.877,Z 1185.149,A -85,B 0,C 180,E1 24764.796,E2 24764.796} C_VEL
LIN {X 0,Y 512.392,Z 1191.067,A -85,B 0,C 180,E1 24762.395,E2 24762.395} C_VEL
LIN {X 0,Y 512.119,Z 1196.106,A -85,B 0,C 180,E1 24759.893,E2 24759.893} C_VEL
LIN {X 0,Y 511.976,Z 1200.316,A -85,B 0,C 180,E1 24757.18,E2 24757.18} C_VEL
LIN {X 0,Y 511.918,Z 1203.42,A -85,B 0,C 180,E1 24754.144,E2 24754.144} C_VEL
LIN {X 0,Y 511.911,Z 1204.713,A -85,B 0,C 180,E1 24751.455,E2 24751.455} C_VEL
LIN {X 0,Y 511.905,Z 1204.826,A -85,B 0,C 180,E1 24749.105,E2 24749.105} C_VEL
LIN {X 0,Y 511.916,Z 1203.964,A -85,B 0,C 180,E1 24746.753,E2 24746.753} C_VEL
LIN {X 0,Y 511.938,Z 1201.971,A -85,B 0,C 180,E1 24744.283,E2 24744.283} C_VEL
LIN {X 0,Y 512.013,Z 1198.878,A -85,B 0,C 180,E1 24741.804,E2 24741.804} C_VEL
LIN {X 0,Y 512.228,Z 1193.819,A -85,B 0,C 180,E1 24738.858,E2 24738.858} C_VEL
LIN {X 0,Y 512.722,Z 1186.966,A -85,B 0,C 180,E1 24735.891,E2 24735.891} C_VEL
LIN {X 0,Y 513.395,Z 1179.855,A -85,B 0,C 180,E1 24733.364,E2 24733.364} C_VEL
LIN {X 0,Y 514.356,Z 1171.888,A -85,B 0,C 180,E1 24730.939,E2 24730.939} C_VEL
LIN {X 0,Y 515.731,Z 1162.227,A -85,B 0,C 180,E1 24728.386,E2 24728.386} C_VEL
LIN {X 0,Y 518.063,Z 1148.281,A -85,B 0,C 180,E1 24725.241,E2 24725.241} C_VEL
LIN {X 0,Y 520.27,Z 1136.354,A -85,B 0,C 180,E1 24722.905,E2 24722.905} C_VEL
LIN {X 0,Y 522.703,Z 1124.354,A -85,B 0,C 180,E1 24720.805,E2 24720.805} C_VEL
LIN {X 0,Y 525.585,Z 1110.559,A -85,B 0,C 180,E1 24718.671,E2 24718.671} C_VEL
LIN {X 0,Y 529.54,Z 1092.29,A -85,B 0,C 180,E1 24716.151,E2 24716.151} C_VEL
LIN {X 0,Y 533.683,Z 1073.474,A -85,B 0,C 180,E1 24713.899,E2 24713.899} C_VEL
LIN {X 0,Y 537.395,Z 1056.869,A -85,B 0,C 180,E1 24712.122,E2 24712.122} C_VEL
LIN {X 0,Y 541.356,Z 1039.091,A -85,B 0,C 180,E1 24710.417,E2 24710.417} C_VEL
LIN {X 0,Y 546.306,Z 1016.556,A -85,B 0,C 180,E1 24708.506,E2 24708.506} C_VEL
LIN {X 0,Y 550.877,Z 994.356,A -85,B 0,C 180,E1 24706.886,E2 24706.886} C_VEL
LIN {X 0,Y 554.552,Z 975.749,A -85,B 0,C 180,E1 24705.688,E2 24705.688} C_VEL
LIN {X 0,Y 558.084,Z 956.651,A -85,B 0,C 180,E1 24704.597,E2 24704.597} C_VEL
LIN {X 0,Y 561.622,Z 936.031,A -85,B 0,C 180,E1 24703.566,E2 24703.566} C_VEL
LIN {X 0,Y 565.54,Z 911.124,A -85,B 0,C 180,E1 24702.503,E2 24702.503} C_VEL
LIN {X 0,Y 569.026,Z 884.681,A -85,B 0,C 180,E1 24701.593,E2 24701.593} C_VEL
LIN {X 0,Y 571.494,Z 862.613,A -85,B 0,C 180,E1 24700.978,E2 24700.978} C_VEL
LIN {X 0,Y 573.489,Z 841.201,A -85,B 0,C 180,E1 24700.503,E2 24700.503} C_VEL
LIN {X 0,Y 575.059,Z 817.644,A -85,B 0,C 180,E1 24700.095,E2 24700.095} C_VEL
LIN {X 0,Y 583.578,Z 597.891,A -85,B 0,C 180,E1 24696.861,E2 24696.861} C_VEL
LIN {X 0,Y 589.884,Z 442.333,A -85,B 0,C 180,E1 24694.533,E2 24694.533} C_VEL
LIN {X 0,Y 578.292,Z 424.41,A -85,B 0,C 180,E1 24692.441,E2 24692.441} C_VEL
LIN {X 0,Y 566.283,Z 406.874,A -85,B 0,C 180,E1 24690.068,E2 24690.068} C_VEL
LIN {X 0,Y 555.155,Z 391.623,A -85,B 0,C 180,E1 24687.632,E2 24687.632} C_VEL
LIN {X 0,Y 546.092,Z 379.776,A -85,B 0,C 180,E1 24685.428,E2 24685.428} C_VEL
LIN {X 0,Y 538.427,Z 370.016,A -85,B 0,C 180,E1 24683.359,E2 24683.359} C_VEL
LIN {X 0,Y 534.581,Z 365.084,A -85,B 0,C 180,E1 24682.228,E2 24682.228} C_VEL
LIN {X 0,Y 530.239,Z 360.01,A -85,B 0,C 180,E1 24680.88,E2 24680.88} C_VEL
LIN {X 0,Y 528.665,Z 358.203,A -85,B 0,C 180,E1 24680.366,E2 24680.366} C_VEL
LIN {X 0,Y 524.495,Z 353.077,A -85,B 0,C 180,E1 24678.91,E2 24678.91} C_VEL
LIN {X 0,Y 521.592,Z 350.562,A -85,B 0,C 180,E1 24677.862,E2 24677.862} C_VEL
LIN {X 0,Y 519.3,Z 346.853,A -85,B 0,C 180,E1 24676.903,E2 24676.903} C_VEL
LIN {X 0,Y 516.001,Z 344.746,A -85,B 0,C 180,E1 24675.568,E2 24675.568} C_VEL
LIN {X 0,Y 514.204,Z 342,A -85,B 0,C 180,E1 24674.7,E2 24674.7} C_VEL
LIN {X 0,Y 513.758,Z 340.17,A -85,B 0,C 180,E1 24674.368,E2 24674.368} C_VEL
LIN {X 0,Y 513.762,Z 340.196,A -85,B 0,C 180,E1 24670.882,E2 24670.882} C_VEL
LIN {X 0,Y 513.812,Z 340.184,A -85,B 0,C 180,E1 24667.492,E2 24667.492} C_VEL
LIN {X 0,Y 513.751,Z 340.175,A -85,B 0,C 180,E1 24664.13,E2 24664.13} C_VEL
LIN {X 0,Y 513.752,Z 340.227,A -85,B 0,C 180,E1 24660.558,E2 24660.558} C_VEL
LIN {X 0,Y 513.794,Z 340.16,A -85,B 0,C 180,E1 24657.211,E2 24657.211} C_VEL
LIN {X 0,Y 513.751,Z 340.238,A -85,B 0,C 180,E1 24653.855,E2 24653.855} C_VEL
LIN {X 0,Y 513.738,Z 340.17,A -85,B 0,C 180,E1 24650.364,E2 24650.364} C_VEL
LIN {X 0,Y 513.795,Z 340.201,A -85,B 0,C 180,E1 24647.068,E2 24647.068} C_VEL
LIN {X 0,Y 513.82,Z 340.35,A -85,B 0,C 180,E1 24645.043,E2 24645.043} C_VEL
LIN {X 0,Y 514.746,Z 343.157,A -85,B 0,C 180,E1 24644.509,E2 24644.509} C_VEL
LIN {X 0,Y 517.023,Z 345.71,A -85,B 0,C 180,E1 24643.484,E2 24643.484} C_VEL
LIN {X 0,Y 519.874,Z 347.305,A -85,B 0,C 180,E1 24642.367,E2 24642.367} C_VEL
LIN {X 0,Y 521.483,Z 350.474,A -85,B 0,C 180,E1 24641.672,E2 24641.672} C_VEL
LIN {X 0,Y 524.686,Z 353.181,A -85,B 0,C 180,E1 24640.519,E2 24640.519} C_VEL
LIN {X 0,Y 525.769,Z 353.872,A -85,B 0,C 180,E1 24640.156,E2 24640.156} C_VEL
LIN {X 0,Y 528.082,Z 357.556,A -85,B 0,C 180,E1 24639.321,E2 24639.321} C_VEL
LIN {X 0,Y 531.503,Z 360.483,A -85,B 0,C 180,E1 24638.247,E2 24638.247} C_VEL
LIN {X 0,Y 534.407,Z 364.54,A -85,B 0,C 180,E1 24637.329,E2 24637.329} C_VEL
LIN {X 0,Y 537.043,Z 366.918,A -85,B 0,C 180,E1 24636.578,E2 24636.578} C_VEL
LIN {X 0,Y 540.377,Z 371.151,A -85,B 0,C 180,E1 24635.63,E2 24635.63} C_VEL
LIN {X 0,Y 542.322,Z 373.139,A -85,B 0,C 180,E1 24635.113,E2 24635.113} C_VEL
LIN {X 0,Y 545.966,Z 377.583,A -85,B 0,C 180,E1 24634.159,E2 24634.159} C_VEL
LIN {X 0,Y 547.789,Z 379.81,A -85,B 0,C 180,E1 24633.698,E2 24633.698} C_VEL
LIN {X 0,Y 552.847,Z 385.858,A -85,B 0,C 180,E1 24632.477,E2 24632.477} C_VEL
LIN {X 0,Y 557.787,Z 391.969,A -85,B 0,C 180,E1 24631.346,E2 24631.346} C_VEL
LIN {X 0,Y 566.092,Z 402.379,A -85,B 0,C 180,E1 24629.57,E2 24629.57} C_VEL
LIN {X 0,Y 576.561,Z 416.202,A -85,B 0,C 180,E1 24627.508,E2 24627.508} C_VEL
LIN {X 0,Y 588.092,Z 432.204,A -85,B 0,C 180,E1 24625.427,E2 24625.427} C_VEL
LIN {X 0,Y 589.787,Z 434.972,A -85,B 0,C 180,E1 24625.129,E2 24625.129} C_VEL
LIN {X 0,Y 581.039,Z 648.374,A -85,B 0,C 180,E1 24621.955,E2 24621.955} C_VEL
LIN {X 0,Y 575.013,Z 799.818,A -85,B 0,C 180,E1 24619.718,E2 24619.718} C_VEL
LIN {X 0,Y 573.235,Z 824.277,A -85,B 0,C 180,E1 24619.257,E2 24619.257} C_VEL
LIN {X 0,Y 570.392,Z 852.348,A -85,B 0,C 180,E1 24618.536,E2 24618.536} C_VEL
LIN {X 0,Y 567.65,Z 874.242,A -85,B 0,C 180,E1 24617.826,E2 24617.826} C_VEL
LIN {X 0,Y 564.803,Z 894.177,A -85,B 0,C 180,E1 24617.055,E2 24617.055} C_VEL
LIN {X 0,Y 562.314,Z 909.896,A -85,B 0,C 180,E1 24616.361,E2 24616.361} C_VEL
LIN {X 0,Y 560.415,Z 917.036,A -85,B 0,C 180,E1 24616.097,E2 24616.097} C_VEL
LIN {X 0,Y 553.012,Z 935.096,A -85,B 0,C 180,E1 24615.617,E2 24615.617} C_VEL
LIN {X 0,Y 550.967,Z 941.891,A -85,B 0,C 180,E1 24615.296,E2 24615.296} C_VEL
LIN {X 0,Y 546.427,Z 963.764,A -85,B 0,C 180,E1 24613.908,E2 24613.908} C_VEL
LIN {X 0,Y 542.36,Z 982.215,A -85,B 0,C 180,E1 24612.577,E2 24612.577} C_VEL
LIN {X 0,Y 538.234,Z 1000.164,A -85,B 0,C 180,E1 24611.118,E2 24611.118} C_VEL
LIN {X 0,Y 533.502,Z 1020.187,A -85,B 0,C 180,E1 24609.281,E2 24609.281} C_VEL
LIN {X 0,Y 528.369,Z 1041.143,A -85,B 0,C 180,E1 24607.058,E2 24607.058} C_VEL
LIN {X 0,Y 524.45,Z 1056.996,A -85,B 0,C 180,E1 24605.153,E2 24605.153} C_VEL
LIN {X 0,Y 521.05,Z 1070.942,A -85,B 0,C 180,E1 24603.286,E2 24603.286} C_VEL
LIN {X 0,Y 517.635,Z 1085.211,A -85,B 0,C 180,E1 24601.16,E2 24601.16} C_VEL
LIN {X 0,Y 513.995,Z 1101.332,A -85,B 0,C 180,E1 24598.443,E2 24598.443} C_VEL
LIN {X 0,Y 510.824,Z 1116.352,A -85,B 0,C 180,E1 24595.507,E2 24595.507} C_VEL
LIN {X 0,Y 508.843,Z 1127.186,A -85,B 0,C 180,E1 24593.127,E2 24593.127} C_VEL
LIN {X 0,Y 506.963,Z 1139.053,A -85,B 0,C 180,E1 24590.145,E2 24590.145} C_VEL
LIN {X 0,Y 505.635,Z 1148.74,A -85,B 0,C 180,E1 24587.228,E2 24587.228} C_VEL
LIN {X 0,Y 504.896,Z 1155.634,A -85,B 0,C 180,E1 24584.801,E2 24584.801} C_VEL
LIN {X 0,Y 504.403,Z 1161.474,A -85,B 0,C 180,E1 24582.362,E2 24582.362} C_VEL
LIN {X 0,Y 504.113,Z 1166.642,A -85,B 0,C 180,E1 24579.706,E2 24579.706} C_VEL
LIN {X 0,Y 503.959,Z 1171.127,A -85,B 0,C 180,E1 24576.608,E2 24576.608} C_VEL
LIN {X 0,Y 503.914,Z 1173.661,A -85,B 0,C 180,E1 24573.754,E2 24573.754} C_VEL
LIN {X 0,Y 503.909,Z 1174.726,A -85,B 0,C 180,E1 24571.364,E2 24571.364} C_VEL
LIN {X 0,Y 503.907,Z 1174.812,A -85,B 0,C 180,E1 24568.977,E2 24568.977} C_VEL
LIN {X 0,Y 503.912,Z 1173.92,A -85,B 0,C 180,E1 24566.587,E2 24566.587} C_VEL
LIN {X 0,Y 503.943,Z 1171.901,A -85,B 0,C 180,E1 24564.078,E2 24564.078} C_VEL
LIN {X 0,Y 504.036,Z 1168.619,A -85,B 0,C 180,E1 24561.444,E2 24561.444} C_VEL
LIN {X 0,Y 504.303,Z 1163.198,A -85,B 0,C 180,E1 24558.333,E2 24558.333} C_VEL
LIN {X 0,Y 504.79,Z 1156.777,A -85,B 0,C 180,E1 24555.548,E2 24555.548} C_VEL
LIN {X 0,Y 505.496,Z 1149.991,A -85,B 0,C 180,E1 24553.096,E2 24553.096} C_VEL
LIN {X 0,Y 506.487,Z 1142.187,A -85,B 0,C 180,E1 24550.675,E2 24550.675} C_VEL
LIN {X 0,Y 507.896,Z 1132.849,A -85,B 0,C 180,E1 24548.157,E2 24548.157} C_VEL
LIN {X 0,Y 510.232,Z 1119.628,A -85,B 0,C 180,E1 24545.082,E2 24545.082} C_VEL
LIN {X 0,Y 513.079,Z 1105.314,A -85,B 0,C 180,E1 24542.222,E2 24542.222} C_VEL
LIN {X 0,Y 516.035,Z 1092.163,A -85,B 0,C 180,E1 24539.879,E2 24539.879} C_VEL
LIN {X 0,Y 520.306,Z 1074.008,A -85,B 0,C 180,E1 24537.055,E2 24537.055} C_VEL
LIN {X 0,Y 524.122,Z 1058.33,A -85,B 0,C 180,E1 24534.928,E2 24534.928} C_VEL
LIN {X 0,Y 527.906,Z 1042.979,A -85,B 0,C 180,E1 24533.063,E2 24533.063} C_VEL
LIN {X 0,Y 531.995,Z 1026.353,A -85,B 0,C 180,E1 24531.255,E2 24531.255} C_VEL
LIN {X 0,Y 537.315,Z 1004.315,A -85,B 0,C 180,E1 24529.15,E2 24529.15} C_VEL
LIN {X 0,Y 541.846,Z 984.597,A -85,B 0,C 180,E1 24527.517,E2 24527.517} C_VEL
LIN {X 0,Y 545.878,Z 966.38,A -85,B 0,C 180,E1 24526.183,E2 24526.183} C_VEL
LIN {X 0,Y 549.572,Z 948.71,A -85,B 0,C 180,E1 24525.031,E2 24525.031} C_VEL
LIN {X 0,Y 553.324,Z 929.394,A -85,B 0,C 180,E1 24523.916,E2 24523.916} C_VEL
LIN {X 0,Y 557.525,Z 905.937,A -85,B 0,C 180,E1 24522.744,E2 24522.744} C_VEL
LIN {X 0,Y 561.535,Z 879.969,A -85,B 0,C 180,E1 24521.673,E2 24521.673} C_VEL
LIN {X 0,Y 564.454,Z 857.96,A -85,B 0,C 180,E1 24520.924,E2 24520.924} C_VEL
LIN {X 0,Y 566.826,Z 836.867,A -85,B 0,C 180,E1 24520.332,E2 24520.332} C_VEL
LIN {X 0,Y 568.834,Z 815.008,A -85,B 0,C 180,E1 24519.843,E2 24519.843} C_VEL
LIN {X 0,Y 570.612,Z 786.936,A -85,B 0,C 180,E1 24519.366,E2 24519.366} C_VEL
LIN {X 0,Y 579.73,Z 563.384,A -85,B 0,C 180,E1 24516.058,E2 24516.058} C_VEL
LIN {X 0,Y 585.074,Z 438.991,A -85,B 0,C 180,E1 24514.186,E2 24514.186} C_VEL
LIN {X 0,Y 572.745,Z 421.641,A -85,B 0,C 180,E1 24511.907,E2 24511.907} C_VEL
LIN {X 0,Y 561.689,Z 407.082,A -85,B 0,C 180,E1 24509.662,E2 24509.662} C_VEL
LIN {X 0,Y 552.569,Z 395.595,A -85,B 0,C 180,E1 24507.626,E2 24507.626} C_VEL
LIN {X 0,Y 548.475,Z 390.585,A -85,B 0,C 180,E1 24506.646,E2 24506.646} C_VEL
LIN {X 0,Y 543.669,Z 384.773,A -85,B 0,C 180,E1 24505.432,E2 24505.432} C_VEL
LIN {X 0,Y 539.825,Z 379.882,A -85,B 0,C 180,E1 24504.397,E2 24504.397} C_VEL
LIN {X 0,Y 535.72,Z 375.42,A -85,B 0,C 180,E1 24503.251,E2 24503.251} C_VEL
LIN {X 0,Y 534.195,Z 373.47,A -85,B 0,C 180,E1 24502.796,E2 24502.796} C_VEL
LIN {X 0,Y 530.517,Z 369.531,A -85,B 0,C 180,E1 24501.679,E2 24501.679} C_VEL
LIN {X 0,Y 529.122,Z 367.476,A -85,B 0,C 180,E1 24501.216,E2 24501.216} C_VEL
LIN {X 0,Y 525.501,Z 364.074,A -85,B 0,C 180,E1 24500.029,E2 24500.029} C_VEL
LIN {X 0,Y 523.825,Z 361.243,A -85,B 0,C 180,E1 24499.399,E2 24499.399} C_VEL
LIN {X 0,Y 520.176,Z 358.46,A -85,B 0,C 180,E1 24498.086,E2 24498.086} C_VEL
LIN {X 0,Y 518.182,Z 355.009,A -85,B 0,C 180,E1 24497.23,E2 24497.23} C_VEL
LIN {X 0,Y 514.196,Z 352.144,A -85,B 0,C 180,E1 24495.566,E2 24495.566} C_VEL
LIN {X 0,Y 512.496,Z 349.111,A -85,B 0,C 180,E1 24494.693,E2 24494.693} C_VEL
LIN {X 0,Y 512.131,Z 348.006,A -85,B 0,C 180,E1 24494.472,E2 24494.472} C_VEL
LIN {X 0,Y 508.626,Z 346.328,A -85,B 0,C 180,E1 24492.719,E2 24492.719} C_VEL
LIN {X 0,Y 506.569,Z 343.755,A -85,B 0,C 180,E1 24491.442,E2 24491.442} C_VEL
LIN {X 0,Y 505.845,Z 341.183,A -85,B 0,C 180,E1 24490.774,E2 24490.774} C_VEL
LIN {X 0,Y 505.808,Z 341.172,A -85,B 0,C 180,E1 24487.383,E2 24487.383} C_VEL
LIN {X 0,Y 505.797,Z 341.166,A -85,B 0,C 180,E1 24483.967,E2 24483.967} C_VEL
LIN {X 0,Y 505.864,Z 341.189,A -85,B 0,C 180,E1 24480.566,E2 24480.566} C_VEL
LIN {X 0,Y 505.815,Z 341.153,A -85,B 0,C 180,E1 24477.167,E2 24477.167} C_VEL
LIN {X 0,Y 505.814,Z 341.224,A -85,B 0,C 180,E1 24473.644,E2 24473.644} C_VEL
LIN {X 0,Y 505.858,Z 341.148,A -85,B 0,C 180,E1 24470.328,E2 24470.328} C_VEL
LIN {X 0,Y 505.838,Z 341.357,A -85,B 0,C 180,E1 24469.58,E2 24469.58} C_VEL
LIN {X 0,Y 506.674,Z 343.886,A -85,B 0,C 180,E1 24468.906,E2 24468.906} C_VEL
LIN {X 0,Y 509.147,Z 346.761,A -85,B 0,C 180,E1 24467.409,E2 24467.409} C_VEL
LIN {X 0,Y 512.187,Z 348.286,A -85,B 0,C 180,E1 24465.905,E2 24465.905} C_VEL
LIN {X 0,Y 513.658,Z 351.389,A -85,B 0,C 180,E1 24465.111,E2 24465.111} C_VEL
LIN {X 0,Y 516.864,Z 354.209,A -85,B 0,C 180,E1 24463.709,E2 24463.709} C_VEL
LIN {X 0,Y 518.21,Z 355.021,A -85,B 0,C 180,E1 24463.176,E2 24463.176} C_VEL
LIN {X 0,Y 520.615,Z 358.926,A -85,B 0,C 180,E1 24462.161,E2 24462.161} C_VEL
LIN {X 0,Y 523.502,Z 361.49,A -85,B 0,C 180,E1 24461.11,E2 24461.11} C_VEL
LIN {X 0,Y 528.511,Z 367.651,A -85,B 0,C 180,E1 24459.368,E2 24459.368} C_VEL
LIN {X 0,Y 533.025,Z 373.159,A -85,B 0,C 180,E1 24457.936,E2 24457.936} C_VEL
LIN {X 0,Y 538.156,Z 379.664,A -85,B 0,C 180,E1 24456.426,E2 24456.426} C_VEL
LIN {X 0,Y 545.675,Z 389.323,A -85,B 0,C 180,E1 24454.406,E2 24454.406} C_VEL
LIN {X 0,Y 554.746,Z 401.523,A -85,B 0,C 180,E1 24452.2,E2 24452.2} C_VEL
LIN {X 0,Y 563.921,Z 414.326,A -85,B 0,C 180,E1 24450.175,E2 24450.175} C_VEL
LIN {X 0,Y 574.658,Z 430.166,A -85,B 0,C 180,E1 24448.006,E2 24448.006} C_VEL
LIN {X 0,Y 584.061,Z 444.837,A -85,B 0,C 180,E1 24446.252,E2 24446.252} C_VEL
LIN {X 0,Y 585.235,Z 446.971,A -85,B 0,C 180,E1 24446.037,E2 24446.037} C_VEL
LIN {X 0,Y 576.085,Z 663.729,A -85,B 0,C 180,E1 24442.798,E2 24442.798} C_VEL
LIN {X 0,Y 569.556,Z 823.843,A -85,B 0,C 180,E1 24440.421,E2 24440.421} C_VEL
LIN {X 0,Y 567.576,Z 849.49,A -85,B 0,C 180,E1 24439.945,E2 24439.945} C_VEL
LIN {X 0,Y 564.549,Z 877.368,A -85,B 0,C 180,E1 24439.236,E2 24439.236} C_VEL
LIN {X 0,Y 561.702,Z 899.132,A -85,B 0,C 180,E1 24438.538,E2 24438.538} C_VEL
LIN {X 0,Y 558.602,Z 919.93,A -85,B 0,C 180,E1 24437.743,E2 24437.743} C_VEL
LIN {X 0,Y 555.132,Z 940.823,A -85,B 0,C 180,E1 24436.808,E2 24436.808} C_VEL
LIN {X 0,Y 550.489,Z 966.308,A -85,B 0,C 180,E1 24435.471,E2 24435.471} C_VEL
LIN {X 0,Y 545.824,Z 989.258,A -85,B 0,C 180,E1 24434.041,E2 24434.041} C_VEL
LIN {X 0,Y 541.623,Z 1008.865,A -85,B 0,C 180,E1 24432.648,E2 24432.648} C_VEL
LIN {X 0,Y 537.306,Z 1028.271,A -85,B 0,C 180,E1 24431.09,E2 24431.09} C_VEL
LIN {X 0,Y 532.133,Z 1050.969,A -85,B 0,C 180,E1 24429.01,E2 24429.01} C_VEL
LIN {X 0,Y 527.627,Z 1070.111,A -85,B 0,C 180,E1 24426.989,E2 24426.989} C_VEL
LIN {X 0,Y 523.953,Z 1085.848,A -85,B 0,C 180,E1 24425.132,E2 24425.132} C_VEL
LIN {X 0,Y 520.538,Z 1100.664,A -85,B 0,C 180,E1 24423.191,E2 24423.191} C_VEL
LIN {X 0,Y 516.764,Z 1117.582,A -85,B 0,C 180,E1 24420.717,E2 24420.717} C_VEL
LIN {X 0,Y 513.358,Z 1133.698,A -85,B 0,C 180,E1 24417.995,E2 24417.995} C_VEL
LIN {X 0,Y 511.115,Z 1144.874,A -85,B 0,C 180,E1 24415.855,E2 24415.855} C_VEL
LIN {X 0,Y 509.089,Z 1155.766,A -85,B 0,C 180,E1 24413.497,E2 24413.497} C_VEL
LIN {X 0,Y 507.477,Z 1165.432,A -85,B 0,C 180,E1 24411.134,E2 24411.134} C_VEL
LIN {X 0,Y 506.058,Z 1175.533,A -85,B 0,C 180,E1 24408.309,E2 24408.309} C_VEL
LIN {X 0,Y 504.987,Z 1184.843,A -85,B 0,C 180,E1 24405.15,E2 24405.15} C_VEL
LIN {X 0,Y 504.432,Z 1191.064,A -85,B 0,C 180,E1 24402.594,E2 24402.594} C_VEL
LIN {X 0,Y 504.136,Z 1196.103,A -85,B 0,C 180,E1 24400.051,E2 24400.051} C_VEL
LIN {X 0,Y 503.987,Z 1200.154,A -85,B 0,C 180,E1 24397.409,E2 24397.409} C_VEL
LIN {X 0,Y 503.919,Z 1203.349,A -85,B 0,C 180,E1 24394.324,E2 24394.324} C_VEL
LIN {X 0,Y 503.908,Z 1204.69,A -85,B 0,C 180,E1 24391.592,E2 24391.592} C_VEL
LIN {X 0,Y 503.901,Z 1204.848,A -85,B 0,C 180,E1 24389.204,E2 24389.204} C_VEL
LIN {X 0,Y 503.916,Z 1204.029,A -85,B 0,C 180,E1 24386.815,E2 24386.815} C_VEL
LIN {X 0,Y 503.935,Z 1202.196,A -85,B 0,C 180,E1 24384.421,E2 24384.421} C_VEL
LIN {X 0,Y 504.008,Z 1199.354,A -85,B 0,C 180,E1 24382.018,E2 24382.018} C_VEL
LIN {X 0,Y 504.167,Z 1195.483,A -85,B 0,C 180,E1 24379.603,E2 24379.603} C_VEL
LIN {X 0,Y 504.523,Z 1190.047,A -85,B 0,C 180,E1 24376.943,E2 24376.943} C_VEL
LIN {X 0,Y 505.268,Z 1181.973,A -85,B 0,C 180,E1 24373.798,E2 24373.798} C_VEL
LIN {X 0,Y 506.326,Z 1173.402,A -85,B 0,C 180,E1 24371.073,E2 24371.073} C_VEL
LIN {X 0,Y 507.614,Z 1164.519,A -85,B 0,C 180,E1 24368.63,E2 24368.63} C_VEL
LIN {X 0,Y 509.278,Z 1154.743,A -85,B 0,C 180,E1 24366.267,E2 24366.267} C_VEL
LIN {X 0,Y 511.858,Z 1141.399,A -85,B 0,C 180,E1 24363.428,E2 24363.428} C_VEL
LIN {X 0,Y 514.92,Z 1126.078,A -85,B 0,C 180,E1 24360.679,E2 24360.679} C_VEL
LIN {X 0,Y 517.792,Z 1112.88,A -85,B 0,C 180,E1 24358.576,E2 24358.576} C_VEL
LIN {X 0,Y 520.928,Z 1098.946,A -85,B 0,C 180,E1 24356.574,E2 24356.574} C_VEL
LIN {X 0,Y 524.6,Z 1083.083,A -85,B 0,C 180,E1 24354.524,E2 24354.524} C_VEL
LIN {X 0,Y 529.515,Z 1062.038,A -85,B 0,C 180,E1 24352.122,E2 24352.122} C_VEL
LIN {X 0,Y 534.042,Z 1042.511,A -85,B 0,C 180,E1 24350.185,E2 24350.185} C_VEL
LIN {X 0,Y 538.161,Z 1024.469,A -85,B 0,C 180,E1 24348.592,E2 24348.592} C_VEL
LIN {X 0,Y 542.629,Z 1004.379,A -85,B 0,C 180,E1 24347.016,E2 24347.016} C_VEL
LIN {X 0,Y 547.965,Z 979.015,A -85,B 0,C 180,E1 24345.299,E2 24345.299} C_VEL
LIN {X 0,Y 551.971,Z 958.3,A -85,B 0,C 180,E1 24344.091,E2 24344.091} C_VEL
LIN {X 0,Y 555.604,Z 938.034,A -85,B 0,C 180,E1 24343.061,E2 24343.061} C_VEL
LIN {X 0,Y 559.003,Z 917.311,A -85,B 0,C 180,E1 24342.15,E2 24342.15} C_VEL
LIN {X 0,Y 562.557,Z 893.139,A -85,B 0,C 180,E1 24341.252,E2 24341.252} C_VEL
LIN {X 0,Y 565.917,Z 865.322,A -85,B 0,C 180,E1 24340.435,E2 24340.435} C_VEL
LIN {X 0,Y 568.105,Z 843.041,A -85,B 0,C 180,E1 24339.928,E2 24339.928} C_VEL
LIN {X 0,Y 569.712,Z 820.801,A -85,B 0,C 180,E1 24339.531,E2 24339.531} C_VEL
LIN {X 0,Y 578.418,Z 606.227,A -85,B 0,C 180,E1 24336.351,E2 24336.351} C_VEL
LIN {X 0,Y 585.171,Z 446.642,A -85,B 0,C 180,E1 24333.955,E2 24333.955} C_VEL
LIN {X 0,Y 575.074,Z 430.81,A -85,B 0,C 180,E1 24332.085,E2 24332.085} C_VEL
LIN {X 0,Y 563.431,Z 413.609,A -85,B 0,C 180,E1 24329.737,E2 24329.737} C_VEL
LIN {X 0,Y 552.441,Z 398.402,A -85,B 0,C 180,E1 24327.282,E2 24327.282} C_VEL
LIN {X 0,Y 543.696,Z 386.809,A -85,B 0,C 180,E1 24325.111,E2 24325.111} C_VEL
LIN {X 0,Y 536.222,Z 377.204,A -85,B 0,C 180,E1 24323.053,E2 24323.053} C_VEL
LIN {X 0,Y 531.678,Z 371.492,A -85,B 0,C 180,E1 24321.688,E2 24321.688} C_VEL
LIN {X 0,Y 527.868,Z 366.66,A -85,B 0,C 180,E1 24320.456,E2 24320.456} C_VEL
LIN {X 0,Y 522.641,Z 360.611,A -85,B 0,C 180,E1 24318.633,E2 24318.633} C_VEL
LIN {X 0,Y 519.675,Z 357.738,A -85,B 0,C 180,E1 24317.525,E2 24317.525} C_VEL
LIN {X 0,Y 517.799,Z 354.634,A -85,B 0,C 180,E1 24316.722,E2 24316.722} C_VEL
LIN {X 0,Y 514.43,Z 352.308,A -85,B 0,C 180,E1 24315.328,E2 24315.328} C_VEL
LIN {X 0,Y 512.511,Z 349.264,A -85,B 0,C 180,E1 24314.375,E2 24314.375} C_VEL
LIN {X 0,Y 512.098,Z 348,A -85,B 0,C 180,E1 24314.127,E2 24314.127} C_VEL
LIN {X 0,Y 508.368,Z 346.132,A -85,B 0,C 180,E1 24312.264,E2 24312.264} C_VEL
LIN {X 0,Y 506.278,Z 343.019,A -85,B 0,C 180,E1 24310.929,E2 24310.929} C_VEL
LIN {X 0,Y 505.814,Z 341.171,A -85,B 0,C 180,E1 24310.478,E2 24310.478} C_VEL
LIN {X 0,Y 505.839,Z 341.19,A -85,B 0,C 180,E1 24307.04,E2 24307.04} C_VEL
LIN {X 0,Y 505.837,Z 341.152,A -85,B 0,C 180,E1 24303.74,E2 24303.74} C_VEL
LIN {X 0,Y 505.81,Z 341.222,A -85,B 0,C 180,E1 24300.34,E2 24300.34} C_VEL
LIN {X 0,Y 505.836,Z 341.148,A -85,B 0,C 180,E1 24296.941,E2 24296.941} C_VEL
LIN {X 0,Y 505.834,Z 341.213,A -85,B 0,C 180,E1 24293.531,E2 24293.531} C_VEL
LIN {X 0,Y 505.792,Z 341.161,A -85,B 0,C 180,E1 24290.096,E2 24290.096} C_VEL
LIN {X 0,Y 505.875,Z 341.385,A -85,B 0,C 180,E1 24288.918,E2 24288.918} C_VEL
LIN {X 0,Y 506.674,Z 343.985,A -85,B 0,C 180,E1 24288.272,E2 24288.272} C_VEL
LIN {X 0,Y 508.894,Z 346.519,A -85,B 0,C 180,E1 24286.941,E2 24286.941} C_VEL
LIN {X 0,Y 512.217,Z 348.284,A -85,B 0,C 180,E1 24285.299,E2 24285.299} C_VEL
LIN {X 0,Y 513.637,Z 351.418,A -85,B 0,C 180,E1 24284.532,E2 24284.532} C_VEL
LIN {X 0,Y 516.337,Z 353.929,A -85,B 0,C 180,E1 24283.345,E2 24283.345} C_VEL
LIN {X 0,Y 518.161,Z 354.973,A -85,B 0,C 180,E1 24282.625,E2 24282.625} C_VEL
